		(*-----------------------Weiterschaltbedingungen----------------------------*)
		IF fb_bbgen_xml_file.fertig_lesen  AND NOT fb_state_entry.E THEN
			fb_state_entry.i16_next_step := 320;
		ELSIF fb_bbgen_xml_file.bError THEN
			sm_fehler_lesen_band := TRUE;
			fb_state_entry.i16_next_step := FEHLER;
		END_IF

(*=======================================================*)
	320:
		IF fb_state_entry.E THEN
			gst_datensatz_copy.st_band:= gst_datensatz.st_band ;
			fb_bbgen_xml_file.start_lesen_band := FALSE;
		END_IF

		(*-----------------------Weiterschaltbedingungen----------------------------*)
		IF hm_alle_daten_laden THEN
			fb_state_entry.i16_next_step := 350;
		ELSE
			IF gst_datensatz_copy.st_md.s_aktuelles_band<>gst_datensatz.st_md.s_aktuelles_band THEN
				fb_state_entry.i16_next_step := 880;
			ELSE
				fb_state_entry.i16_next_step := 999;
			END_IF
		END_IF

(*=======================================================*)
	350:	(* Wt Daten *)
		IF fb_state_entry.E THEN
			gst_datensatz.st_wt:=st_wt_leer;
		END_IF

		(*-----------------------Weiterschaltbedingungen----------------------------*)
		IF 	gst_datensatz.st_md.s_aktueller_wt <>'' THEN
			fb_state_entry.i16_next_step := 360;
		ELSIF 	hm_alle_daten_laden  THEN
				fb_state_entry.i16_next_step := 400;
			ELSE
				fb_state_entry.i16_next_step := 999;
		END_IF

	360:
		IF fb_state_entry.E THEN
			fb_bbgen_xml_file.start_lesen_wt := TRUE;
			fb_bbgen_xml_file.s_path := s_wt_path;
			fb_bbgen_xml_file.s_wt := gst_datensatz.st_md.s_aktueller_wt;
		END_IF

		(*-----------------------Weiterschaltbedingungen----------------------------*)
		IF fb_bbgen_xml_file.fertig_lesen  AND NOT fb_state_entry.E THEN
			fb_state_entry.i16_next_step := 370;
		ELSIF fb_bbgen_xml_file.bError THEN
			sm_fehler_lesen_wt := TRUE;
			fb_state_entry.i16_next_step := FEHLER;
		END_IF

(*=======================================================*)
	370:
		IF fb_state_entry.E THEN
			gst_datensatz_copy.st_wt:= gst_datensatz.st_wt ;
			fb_bbgen_xml_file.start_lesen_wt := FALSE;
		END_IF

		(*-----------------------Weiterschaltbedingungen----------------------------*)
		IF hm_alle_daten_laden THEN
			fb_state_entry.i16_next_step := 400;
		ELSE
			IF gst_datensatz_copy.st_md.s_aktueller_wt<>gst_datensatz.st_md.s_aktueller_wt THEN
				fb_state_entry.i16_next_step := 880;
			ELSE
				fb_state_entry.i16_next_step := 999;
			END_IF
		END_IF

(*=======================================================*)
	400:	(* Abfrage auf manuelle Anwahl des Bestückbildes *)
 		CASE gst_datensatz.st_md.i16_typ_bestueckmodus OF

			BESTUECKUNG_MANUAL:
				(* Bei der manuellen Auswahl des Bestückprogrammes werden die Daten direkt über die Visu
				von einem txt-File in die Variable "gst_datensatz" geladen. Ein Einlesen ist somit nicht nötig. *)
				gst_datensatz.st_bestueckprogramm:=gst_manuelles_bestueckprogramm;
				gst_datensatz.st_md.s_aktueller_isk:='ISK_Daten';
				IF hm_alle_daten_laden THEN
					fb_state_entry.i16_next_step := 600;
				ELSE
					fb_state_entry.i16_next_step := 999;
				END_IF

			BESTUECKUNG_HALBAUTO:
				IF gi16_maschinenstatusinfo = STATUS_MASCHINE_ARBEITET THEN
					gst_datensatz.st_md.s_aktueller_isk:='ISK_Daten';
					fb_state_entry.i16_next_step := 500;
				ELSE
					fb_state_entry.i16_next_step := 999;
				END_IF

			BESTUECKUNG_AUTO:
				IF gi16_maschinenstatusinfo = STATUS_MASCHINE_ARBEITET THEN
					fb_state_entry.i16_next_step := 410;
				ELSE
					fb_state_entry.i16_next_step := 999;
				END_IF

		END_CASE

(*=======================================================*)
	410:	(*alle Positonen löschen*)
		IF 	fb_state_entry.E THEN
			gst_bestueckbild := st_bestueckbild_leer;
			gst_datensatz.st_bestueckprogramm:=st_bestueckprogramm_leer;
		END_IF

		fb_state_entry.i16_next_step := 412;

(*=======================================================*)
	412:	(* Bestueckbild lesen und generieren *)
		IF fb_state_entry.E THEN
			fb_bbgen_xml_file.start_lesen_bestueckbild := TRUE;
			fb_bbgen_xml_file.s_path := s_bestueckbild_path;
			fb_bbgen_xml_file.s_bestueckbild := gst_datensatz.st_md.s_aktuelle_artikelnummer;
		END_IF

		(*-----------------------Weiterschaltbedingungen----------------------------*)
		IF fb_bbgen_xml_file.fertig_lesen  AND NOT fb_state_entry.E THEN
			IF	visu.b_merker_vollbestuecken THEN
				fb_state_entry.i16_next_step := 414;
			ELSE
				fb_state_entry.i16_next_step := 420;
			END_IF
		ELSIF fb_bbgen_xml_file.bError THEN
			sm_fehler_lesen_bestueckbild := TRUE;
			fb_state_entry.i16_next_step := FEHLER;
		END_IF

(*=======================================================*)
	414:	(* Werkzeuggruppen durchsuchen nach benuztem Werkzeug *)
		IF 	fb_state_entry.E THEN
			fb_bbgen_xml_file.start_lesen_bestueckbild := FALSE;
			i32_UsedTool:=-1;
			k:=-1;
			FOR k := 0 TO 4 DO
				i:=-1;

				FOR i := 0 TO MaxNoOfWkz DO
					IF 	gst_bestueckbild.s_wkzgruppe[k].s_wkznummer[i] = gst_datensatz.st_md.s_aktuelles_wkz THEN
						i32_UsedTool:=i;
					END_IF
				END_FOR
			END_FOR
		END_IF

		(*-----------------------Weiterschaltbedingungen----------------------------*)
		IF 	i32_UsedTool <> -1 THEN
			fb_state_entry.i16_next_step := 416;
		END_IF

		IF 	gst_bestueckbild.s_Bestueckbild_vollbestueckt[i32_UsedTool] = '' THEN
			fb_state_entry.i16_next_step := 420;
			bm_keine_vollbestueck_Artikelnummer:=TRUE;
		END_IF

(*=======================================================*)
	416:	(* Bestueckbild lesen und generieren *)
		IF fb_state_entry.E THEN
			fb_bbgen_xml_file.start_lesen_bestueckbild := TRUE;
			fb_bbgen_xml_file.s_path := s_bestueckbild_path;
			fb_bbgen_xml_file.s_bestueckbild := gst_bestueckbild.s_Bestueckbild_vollbestueckt[i32_UsedTool] ;
		END_IF

		(*-----------------------Weiterschaltbedingungen----------------------------*)
		IF fb_bbgen_xml_file.fertig_lesen  AND NOT fb_state_entry.E THEN
			fb_state_entry.i16_next_step := 420;
			fb_bbgen_xml_file.start_lesen_bestueckbild := FALSE;
		ELSIF fb_bbgen_xml_file.bError THEN
			sm_fehler_lesen_bestueckbild := TRUE;
			fb_state_entry.i16_next_step := FEHLER;
		END_IF

(*=======================================================*)
	420:	(* Generiere Bestückprogramm *)
		IF fb_state_entry.E THEN
			bm_kleinster_greifer_groesser_kleinste_pinanzahl_in_bb := FALSE;
			generiere_bestueckbild();
		END_IF

		(*-----------------------Weiterschaltbedingungen----------------------------*)
		fb_state_entry.i16_next_step := 425;

(*=======================================================*)
	425:	(* Hub_Faktor_ermitteln *)
		IF fb_state_entry.E THEN

			IF	gst_datensatz.st_wkz.i16_typ_bandeinzug=STANDARD_2FACH_V2  OR
				gst_datensatz.st_wkz.i16_typ_bandeinzug=BANDWECHSLER_V2 THEN
				Hub_Faktor_ermitteln();
			ELSE
				lr_FaktorHub:=1;
			END_IF

		END_IF

		(*-----------------------Weiterschaltbedingungen----------------------------*)
		fb_state_entry.i16_next_step := 430;

(*=======================================================*)
	430:	(* Schreibe Bestückprogramm auf HDD *)
		IF fb_state_entry.E THEN
			fb_bbgen_write_file.bStart := TRUE;
		END_IF


		(*-----------------------Weiterschaltbedingungen----------------------------*)
		IF NOT fb_state_entry.E THEN
			IF fb_bbgen_write_file.bFertig THEN
				fb_state_entry.i16_next_step := 600; (* ISK Daten lesen*)
			END_IF

			IF fb_bbgen_write_file.bError THEN
				fb_state_entry.i16_next_step := FEHLER;
				sm_fehler_schreiben_bestueckbild_auf_hdd := TRUE;
			END_IF
		END_IF

		IF fb_state_entry.X THEN
			fb_bbgen_write_file.bStart := FALSE;
		END_IF


(*=======================================================*)
	500:	(*alle Positonen löschen*)
		IF 	fb_state_entry.E THEN
			gst_bestueckbild_halbauto := st_bestueckbild_halbauto_leer;
		END_IF

		fb_state_entry.i16_next_step := 510;

(*=======================================================*)
	510:	(* halbauto Bestueckbild lesen  *)
		IF fb_state_entry.E THEN
			fb_bbgen_xml_file.start_lesen_bestueckbild_halbauto := TRUE;
			fb_bbgen_xml_file.s_path := s_bestueckbild_halbauto_path;
			fb_bbgen_xml_file.s_bestueckbild := gst_datensatz.st_md.s_aktuelle_artikelnummer;
		END_IF

		(*-----------------------Weiterschaltbedingungen----------------------------*)
		IF fb_bbgen_xml_file.fertig_lesen  AND NOT fb_state_entry.E THEN
			fb_state_entry.i16_next_step := 515;
		ELSIF fb_bbgen_xml_file.bError THEN
			sm_fehler_lesen_bestueckbild := TRUE;
			fb_state_entry.i16_next_step := FEHLER;
		END_IF

(*=======================================================*)
	515:	(* alle Positionen löschen  *)
		fb_bbgen_xml_file.start_lesen_bestueckbild_halbauto := FALSE;
		gst_datensatz.st_bestueckprogramm:=st_bestueckprogramm_leer;

		(*-----------------------Weiterschaltbedingungen----------------------------*)
		IF	b_Wkz_Gruppe_gebildet THEN
			fb_state_entry.i16_next_step := 540;
		ELSE
			fb_state_entry.i16_next_step := 520;
		END_IF

		IF	sm_Wkz_nicht_kompatibel OR
			sm_Wkz_Gruppe_nicht_zugeordnet THEN
			fb_state_entry.i16_next_step := FEHLER;
		END_IF

(*=======================================================*)
	520:	(* Werkzeuggruppen durchsuchen nach benuztem Werkzeug *)
		IF 	fb_state_entry.E THEN
			i32_UsedTool:=-1;
			k:=-1;
			FOR k := 0 TO 4 DO
				i:=-1;

				FOR i := 0 TO MaxNoOfWkz DO
					IF 	gst_bestueckbild_halbauto.s_wkzgruppe[k].s_wkznummer[i] = gst_datensatz.st_md.s_aktuelles_wkz THEN
						i32_UsedTool:=i;
					END_IF
				END_FOR
			END_FOR

		END_IF

		(*-----------------------Weiterschaltbedingungen----------------------------*)
		IF 	i32_UsedTool <> -1 THEN
			fb_state_entry.i16_next_step := 530;
		ELSE
			sm_fehler_wkz_nicht_vorhanden:=TRUE;
			fb_state_entry.i16_next_step := FEHLER;
		END_IF

(*=======================================================*)
	530: (*kopieren des zum WZ passenden Bestückbild*)
		IF 	fb_state_entry.E THEN
			gst_datensatz.st_bestueckprogramm:=gst_bestueckbild_halbauto.Wkz[i32_UsedTool];
			gst_datensatz.st_isk:=gst_bestueckbild_halbauto.Wkz[i32_UsedTool].st_isk;


			(*Offset dazurechnen*)
			k:=-1;
			FOR k := 0 TO (gst_bestueckbild_halbauto.Wkz[i32_UsedTool].i32_anzahl - 1) DO  (*max 511*)
				IF	gst_datensatz.st_bestueckprogramm.i16_b[k] = -1 THEN
					gst_datensatz.st_bestueckprogramm.lr_y[k]:=gst_datensatz.st_bestueckprogramm.lr_y[k] + gst_datensatz.st_bestueckprogramm.lr_y_offset;
					gst_datensatz.st_bestueckprogramm.lr_z[k]:=gst_datensatz.st_bestueckprogramm.lr_z[k] + gst_datensatz.st_bestueckprogramm.lr_z_offset;
				END_IF
			END_FOR

		END_IF

		(*-----------------------Weiterschaltbedingungen----------------------------*)
		IF 	gst_datensatz.st_bestueckprogramm.s_band = gst_datensatz.st_md.s_aktuelles_band  THEN
			fb_state_entry.i16_next_step := 590;
		ELSE
			sm_fehler_falsches_Band:=TRUE;
			fb_state_entry.i16_next_step := FEHLER;
		END_IF

(*=======================================================*)
(*Halbautomatisch mit Gruppen*)
	540:	(* prüfen ob Werkzeuggruppen gleiche Bänder haben *)
		IF 	fb_state_entry.E THEN

			k:=-1;
			FOR k := 0 TO 4 DO
				i:=-1;

				FOR i := 0 TO MaxNoOfWkz DO
					n:=-1;
					FOR n := 0 TO i16_anzahl_Wkz_Gruppen - 1 DO
						IF 	gst_bestueckbild_halbauto.s_wkzgruppe[k].s_wkznummer[i] = gst_datensatz.st_md.st_wkz_gruppe[n].s_wkz THEN
							gst_datensatz.st_md.st_wkz_gruppe[n].s_Band:=gst_bestueckbild_halbauto.Wkz[i].s_band;
							gst_datensatz.st_md.st_wkz_gruppe[n].i32_Anzahl:=gst_bestueckbild_halbauto.Wkz[i].i32_anzahl;
							gst_datensatz.st_md.st_wkz_gruppe[n].i32_Wkz_nr:=i;
						END_IF
					END_FOR

				END_FOR

			END_FOR

		END_IF


		i:=-1;
		b_Wkz_akt_vorhanden:=FALSE;
		FOR i := 0 TO i16_anzahl_Wkz_Gruppen - 1 DO
			IF	gst_datensatz.st_md.st_wkz_gruppe[i].s_Band <> '' AND
				gst_datensatz.st_md.st_wkz_gruppe[0].s_Band <> gst_datensatz.st_md.st_wkz_gruppe[i].s_Band THEN
				sm_Band_nicht_kompatibel:=TRUE;
			END_IF
			IF	gst_datensatz.st_md.s_aktuelles_wkz = gst_datensatz.st_md.st_wkz_gruppe[i].s_wkz THEN
				b_Wkz_akt_vorhanden:=TRUE;
			END_IF
		END_FOR
		sm_fehler_wkz_nicht_vorhanden:=NOT b_Wkz_akt_vorhanden;

		(*-----------------------Weiterschaltbedingungen----------------------------*)
		IF	sm_fehler_wkz_nicht_vorhanden OR
			sm_Band_nicht_kompatibel THEN
			fb_state_entry.i16_next_step := FEHLER;
		ELSE
			fb_state_entry.i16_next_step := 550;
		END_IF

(*=======================================================*)
	550: (*kopieren des zum WZ passenden Bestückbild*)
		IF 	fb_state_entry.E THEN
			i32_UsedTool:=gst_datensatz.st_md.st_wkz_gruppe[0].i32_Wkz_nr;
			gst_datensatz.st_bestueckprogramm:=gst_bestueckbild_halbauto.Wkz[i32_UsedTool];
			gst_datensatz.st_isk:=gst_bestueckbild_halbauto.Wkz[i32_UsedTool].st_isk;
			gst_datensatz.st_bestueckprogramm.i32_anzahl:=0;

			i:=-1;
			for_begin:=0;
			FOR i := 0 TO i16_anzahl_Wkz_Gruppen - 1 DO

				i32_UsedTool:=gst_datensatz.st_md.st_wkz_gruppe[i].i32_Wkz_nr;
				gst_datensatz.st_bestueckprogramm.i32_anzahl:=gst_datensatz.st_md.st_wkz_gruppe[i].i32_Anzahl + gst_datensatz.st_bestueckprogramm.i32_anzahl;

				for_end:=for_begin + gst_bestueckbild_halbauto.Wkz[i32_UsedTool].i32_anzahl - 1;

				FOR k := for_begin TO for_end DO  (*max 511*)
						gst_datensatz.st_bestueckprogramm.lr_y[k]:=		gst_bestueckbild_halbauto.Wkz[i32_UsedTool].lr_y[k - for_begin] + gst_bestueckbild_halbauto.Wkz[i32_UsedTool].lr_y_offset;
						gst_datensatz.st_bestueckprogramm.lr_z[k]:=		gst_bestueckbild_halbauto.Wkz[i32_UsedTool].lr_z[k - for_begin] + gst_bestueckbild_halbauto.Wkz[i32_UsedTool].lr_z_offset;
						gst_datensatz.st_bestueckprogramm.i16_b[k]:=	gst_bestueckbild_halbauto.Wkz[i32_UsedTool].i16_b[k - for_begin];
						gst_datensatz.st_bestueckprogramm.b_podest_verschieben[k]:=	gst_bestueckbild_halbauto.Wkz[i32_UsedTool].b_podest_verschieben[k - for_begin];
				END_FOR
				for_begin:=for_begin + gst_bestueckbild_halbauto.Wkz[i32_UsedTool].i32_anzahl ;

			END_FOR

		END_IF

		(*-----------------------Weiterschaltbedingungen----------------------------*)
		IF 	gst_datensatz.st_bestueckprogramm.s_band = gst_datensatz.st_md.s_aktuelles_band  THEN
			fb_state_entry.i16_next_step := 590;
		ELSE
			sm_fehler_falsches_Band:=TRUE;
			fb_state_entry.i16_next_step := FEHLER;
		END_IF

(*=======================================================*)
(*=======================================================*)
	590:	(* Hub_Faktor_ermitteln *)
		IF fb_state_entry.E THEN

			IF	gst_datensatz.st_wkz.i16_typ_bandeinzug=STANDARD_2FACH_V2 OR
				gst_datensatz.st_wkz.i16_typ_bandeinzug=BANDWECHSLER_V2 OR
				gst_datensatz.st_wkz.i16_typ_bandeinzug=SERVO THEN
				Hub_Faktor_ermitteln_halbauto();
			ELSE
				lr_FaktorHub:=1;
			END_IF

		END_IF

		(*-----------------------Weiterschaltbedingungen----------------------------*)
		fb_state_entry.i16_next_step := 999;

(*ISK Daten lesen===============================================*)
	600:
		IF fb_state_entry.E THEN
			fb_bbgen_xml_file.start_lesen_bestueckbild := FALSE;
			hm_alle_daten_laden:=FALSE;
		END_IF

		(*-----------------------Weiterschaltbedingungen----------------------------*)
		fb_state_entry.i16_next_step := 610;

(*=======================================================*)
	610:(* ISK Daten *)

		IF fb_state_entry.E THEN
			fb_bbgen_xml_file.start_lesen_isk := TRUE;
			fb_bbgen_xml_file.s_path := s_isk_path;
			fb_bbgen_xml_file.s_isk := gst_datensatz.st_md.s_aktueller_isk;
		END_IF

		(*-----------------------Weiterschaltbedingungen----------------------------*)
		IF fb_bbgen_xml_file.fertig_lesen  AND NOT fb_state_entry.E THEN
			fb_state_entry.i16_next_step := 620;
		ELSIF fb_bbgen_xml_file.bError THEN
			sm_fehler_lesen_isk := TRUE;
			fb_state_entry.i16_next_step := FEHLER;
		END_IF

(*=======================================================*)
	620:
		IF fb_state_entry.E THEN
			gst_datensatz_copy.st_isk:= gst_datensatz.st_isk ;
			fb_bbgen_xml_file.start_lesen_isk := FALSE;
		END_IF

		(*-----------------------Weiterschaltbedingungen----------------------------*)
		fb_state_entry.i16_next_step := 999;




(*===========================Speichern============================*)
	(* Alle aktuelle Daten von der Maschine und Werkzeug speichern *)
	800:	(* ISK daten *)
		IF fb_state_entry.E THEN
			fb_bbgen_xml_file.start_schreiben_isk := TRUE;
			fb_bbgen_xml_file.s_path := s_isk_path;
			fb_bbgen_xml_file.s_isk := gst_datensatz.st_md.s_aktueller_isk;
		END_IF

		(*-----------------------Weiterschaltbedingungen----------------------------*)
		IF fb_bbgen_xml_file.fertig_schreiben AND NOT fb_state_entry.E THEN
			fb_state_entry.i16_next_step := 810;
		ELSIF fb_bbgen_xml_file.bError THEN
			sm_fehler_schreiben_isk := TRUE;
			fb_state_entry.i16_next_step := FEHLER;
		END_IF

(*=======================================================*)
	810:
		IF fb_state_entry.E THEN
			gst_datensatz_copy.st_isk:= gst_datensatz.st_isk ;
			fb_bbgen_xml_file.start_schreiben_isk := FALSE;
		END_IF

		(*-----------------------Weiterschaltbedingungen----------------------------*)
		IF 	hm_alle_daten_speichern THEN
			fb_state_entry.i16_next_step := 820;
		ELSE
			fb_state_entry.i16_next_step := 999;
		END_IF

(*=======================================================*)
	820:	(* WKZ Daten *)
		IF (fb_state_entry.E) THEN
			fb_bbgen_xml_file.start_schreiben_wkz := TRUE;
			fb_bbgen_xml_file.s_path := s_wkz_path;
			fb_bbgen_xml_file.s_wkz := gst_datensatz.st_md.s_aktuelles_wkz;
		END_IF

		(*-----------------------Weiterschaltbedingungen----------------------------*)
		IF fb_bbgen_xml_file.fertig_schreiben  AND NOT fb_state_entry.E THEN
			fb_state_entry.i16_next_step := 830;
		ELSIF fb_bbgen_xml_file.bError THEN
			sm_fehler_schreiben_wkz := TRUE;
			fb_state_entry.i16_next_step := FEHLER;
		END_IF

(*=======================================================*)
	830:
		IF fb_state_entry.E THEN
			fb_bbgen_xml_file.start_schreiben_wkz := FALSE;
			gst_datensatz_copy.st_wkz:= gst_datensatz.st_wkz ;
		END_IF

		(*-----------------------Weiterschaltbedingungen----------------------------*)
		IF 	hm_alle_daten_speichern THEN
			fb_state_entry.i16_next_step := 840;
		ELSE
			fb_state_entry.i16_next_step := 999;
		END_IF

(*=======================================================*)
	840:	(* Band Daten *)
		IF (fb_state_entry.E) THEN
			fb_bbgen_xml_file.start_schreiben_band := TRUE;
			fb_bbgen_xml_file.s_path := s_band_path;
			fb_bbgen_xml_file.s_band := gst_datensatz.st_md.s_aktuelles_band;
		END_IF

		(*-----------------------Weiterschaltbedingungen----------------------------*)
		IF fb_bbgen_xml_file.fertig_schreiben  AND NOT fb_state_entry.E THEN
			fb_state_entry.i16_next_step := 850;
		ELSIF fb_bbgen_xml_file.bError THEN
			sm_fehler_schreiben_band := TRUE;
			fb_state_entry.i16_next_step := FEHLER;
		END_IF

(*=======================================================*)
	850:
		IF fb_state_entry.E THEN
			fb_bbgen_xml_file.start_schreiben_band := FALSE;
			gst_datensatz_copy.st_band:= gst_datensatz.st_band ;
		END_IF

		(*-----------------------Weiterschaltbedingungen----------------------------*)
		IF 	hm_alle_daten_speichern THEN
			fb_state_entry.i16_next_step := 860;
		ELSE
			fb_state_entry.i16_next_step := 999;
		END_IF

(*=======================================================*)
	860:	(* Wt Daten *)
		IF (fb_state_entry.E) THEN
			fb_bbgen_xml_file.start_schreiben_wt := TRUE;
			fb_bbgen_xml_file.s_path := s_wt_path;
			fb_bbgen_xml_file.s_wt := gst_datensatz.st_md.s_aktueller_wt;
		END_IF

		(*-----------------------Weiterschaltbedingungen----------------------------*)
		IF fb_bbgen_xml_file.fertig_schreiben  AND NOT fb_state_entry.E THEN
			fb_state_entry.i16_next_step := 870;
		ELSIF fb_bbgen_xml_file.bError THEN
			sm_fehler_schreiben_wt := TRUE;
			fb_state_entry.i16_next_step := FEHLER;
		END_IF

(*=======================================================*)
	870:
		IF fb_state_entry.E THEN
			fb_bbgen_xml_file.start_schreiben_wt := FALSE;
			gst_datensatz_copy.st_wt:= gst_datensatz.st_wt ;
		END_IF

		(*-----------------------Weiterschaltbedingungen----------------------------*)
		IF 	hm_alle_daten_speichern THEN
			fb_state_entry.i16_next_step := 880;
		ELSE
			fb_state_entry.i16_next_step := 999;
		END_IF

(*=======================================================*)
	880:	(* Maschinendaten *)
		IF (fb_state_entry.E) THEN
			fb_bbgen_xml_file.start_schreiben_md := TRUE;
			fb_bbgen_xml_file.s_path := s_md_path;
			fb_bbgen_xml_file.s_md := s_md_name;
		END_IF

		(*-----------------------Weiterschaltbedingungen----------------------------*)
		IF fb_bbgen_xml_file.fertig_schreiben  AND NOT fb_state_entry.E THEN
			fb_state_entry.i16_next_step := 882;
		ELSIF fb_bbgen_xml_file.bError THEN
			sm_fehler_schreiben_md := TRUE;
			fb_state_entry.i16_next_step := FEHLER;
		END_IF

	882:
		IF fb_state_entry.E THEN
			gst_datensatz_copy.st_md:= gst_datensatz.st_md ;
			fb_bbgen_xml_file.start_schreiben_md := FALSE;
			fb_state_entry.i16_next_step := 884;
		END_IF

	884:	(* Maschinendaten Backup *)
		IF (fb_state_entry.E) THEN
			fb_bbgen_xml_file.start_schreiben_md_backup := TRUE;
			fb_bbgen_xml_file.s_path := s_md_path;
			fb_bbgen_xml_file.s_md_backup := s_md_backup_name;
		END_IF

		(*-----------------------Weiterschaltbedingungen----------------------------*)
		IF fb_bbgen_xml_file.fertig_schreiben  AND NOT fb_state_entry.E THEN
			fb_state_entry.i16_next_step := 886;
		ELSIF fb_bbgen_xml_file.bError THEN
			sm_fehler_schreiben_md := TRUE;
			fb_state_entry.i16_next_step := FEHLER;
		END_IF

	886:
		IF fb_state_entry.E THEN
			fb_bbgen_xml_file.start_schreiben_md_backup := FALSE;
			fb_state_entry.i16_next_step := 999;
		END_IF

(*=======================================================*)
(* manuelle Bestückbilder in halbautomatische XML Dateien umwandeln
	->	PLC resetten (Strukturen leerern)
	->	Artikelnummer in MD eintragen ( Artikelnummer = XML Dateiname)
	->	Schritt 975 forcen
	->	manualle Bestückbilder nacheinader mit Visu vorne öffnen (mit der ersten beginnen)
		die Bestückbilder werden dann in die Struktur (Bestückbild halbauto) eingetragen
	->	Schritt 980 forcen = XML Datei wird erstellt ( D:\BBGen\BestueckbildHalbauto )
	->	in der XML Datei nicht vorhandene WZ löschen, Werkzeuge, Band, Beschreibung, Projekt eintragen
	->	neue XML Datei auf Server kopieren
*)
975:
	IF (fb_state_entry.E) THEN
		gst_manuelles_bestueckprogramm.i32_anzahl:=0;
		gst_manuelles_bestueckprogramm.s_band:='';
		gst_manuelles_bestueckprogramm.lr_y_offset:=0;
		gst_manuelles_bestueckprogramm.lr_z_offset:=0;

		k:=-1;
		FOR k := 0 TO 511 DO
			gst_manuelles_bestueckprogramm.lr_y[k]:=0;
			gst_manuelles_bestueckprogramm.lr_z[k]:=0;
			gst_manuelles_bestueckprogramm.i16_b[k]:=0;
		END_FOR
		gst_manuelles_bestueckprogramm_copy:=gst_manuelles_bestueckprogramm;
		wkz_Nr:=-1;
	END_IF

	fb_ton_wz(IN:= MEMCMP(ADR(gst_manuelles_bestueckprogramm_copy), ADR(gst_manuelles_bestueckprogramm), SIZEOF(gst_manuelles_bestueckprogramm_copy)) <> 0, PT:= t#600ms, Q=> , ET=> );

	IF	fb_ton_wz.Q  THEN
		wkz_Nr:=wkz_Nr+1;
		gst_bestueckbild_halbauto.Wkz[wkz_Nr]:=gst_manuelles_bestueckprogramm;
		gst_bestueckbild_halbauto.Wkz[wkz_Nr].st_isk:=gst_datensatz.st_isk;

		gst_manuelles_bestueckprogramm.i32_anzahl:=0;
		gst_manuelles_bestueckprogramm.s_band:='';
		gst_manuelles_bestueckprogramm.lr_y_offset:=0;
		gst_manuelles_bestueckprogramm.lr_z_offset:=0;

		k:=-1;
		FOR k := 0 TO 511 DO
			gst_manuelles_bestueckprogramm.lr_y[k]:=0;
			gst_manuelles_bestueckprogramm.lr_z[k]:=0;
			gst_manuelles_bestueckprogramm.i16_b[k]:=0;
		END_FOR

		gst_manuelles_bestueckprogramm_copy:=gst_manuelles_bestueckprogramm;
	END_IF

(*=======================================================*)
	980:	(* Bestückbild *)
		IF (fb_state_entry.E) THEN
			fb_bbgen_xml_file.start_schreiben_bestueckbild_halbauto := TRUE;
			fb_bbgen_xml_file.s_path := s_bestueckbild_halbauto_path;
			fb_bbgen_xml_file.s_bestueckbild := gst_datensatz.st_md.s_aktuelle_artikelnummer;
		END_IF

		(*-----------------------Weiterschaltbedingungen----------------------------*)
		IF fb_bbgen_xml_file.fertig_schreiben  AND NOT fb_state_entry.E THEN
			fb_state_entry.i16_next_step := 990;
		ELSIF fb_bbgen_xml_file.bError THEN
			sm_fehler_schreiben_bestueckbild := TRUE;
			fb_state_entry.i16_next_step := FEHLER;
		END_IF

(*=======================================================*)
	990:
		IF fb_state_entry.E THEN
			fb_bbgen_xml_file.start_schreiben_bestueckbild_halbauto := FALSE;
			fb_state_entry.i16_next_step := 999;
		END_IF

(*=======================================================*)
	999:	(* Ende - Befehl wurde korrekt abgearbeitet *)
		IF fb_state_entry.E THEN
			st_ctrl_out.b_fertig := TRUE;
			i16_auftrag := KEIN_BB_AUFTRAG;

			IF NOT b_lesen_komplett THEN
				gst_datensatz_copy := gst_datensatz;
			END_IF
			b_lesen_komplett:=TRUE;

			fb_state_entry.i16_next_step := 0;
		END_IF

(*=======================================================*)
	1000: (* Fehler *)
		IF fb_state_entry.E THEN
			st_ctrl_out.b_fehler := TRUE;
			fb_ton_quitt.IN := FALSE;
			fb_bbgen_xml_file.bQuit := FALSE;
		END_IF

		(*-----------------------Weiterschaltbedingungen----------------------------*)
		IF st_ctrl_in.b_quitt AND NOT fb_state_entry.E THEN
			st_ctrl_out.b_fehler := FALSE;
			fb_ton_quitt.IN := TRUE;
			fb_bbgen_xml_file.bQuit := TRUE;
		END_IF

		IF fb_ton_quitt.Q THEN
			fb_ton_quitt.IN := FALSE;
			fb_state_entry.i16_next_step := 0;
		END_IF
END_CASE

fb_state_entry(	i16_pos:= 2 );

(* ======================================Subkomponenten======================================== *)
fb_bbgen_xml_file(
	bQuit:= ,
	start_lesen_isk:= ,
	start_schreiben_isk:= ,
	start_lesen_wkz:= ,
	start_schreiben_wkz:= ,
	start_lesen_bestueckbild:= ,
	start_schreiben_bestueckbild:= ,
	start_lesen_md:= ,
	start_schreiben_md:= ,
	start_lesen_band:= ,
	start_schreiben_band:= ,
	s_path:= ,
	s_bestueckbild:= ,
	s_wkz:= ,
	s_isk:= ,
	s_md:= ,
	s_band:= ,
	fertig_lesen=> ,
	fertig_schreiben=> ,
	bError=> ,
	nErrId=> );

fb_bbgen_write_file(
	bStart:= ,
	bFertig=> ,
	bError=> );

fb_xml_srv_read(
	sNetId:= ,
	ePath:= PATH_GENERIC,
	nMode:= XMLSRV_SKIPMISSING,
	sSymName:= ,
	sFilePath:= ,
	sXPath:= ,
	bExecute:= ,
	tTimeout:= t#20s,
	bBusy=> ,
	bError=> ,
	nErrId=> );

IF st_config.b_config_fertig THEN
	garr_stoermeldungen[st_config.i16_meld_startindex + 0] := sm_fehler_lesen_band;
	garr_stoermeldungen[st_config.i16_meld_startindex + 1] := sm_fehler_lesen_bestueckbild;
	garr_stoermeldungen[st_config.i16_meld_startindex + 2] := sm_fehler_lesen_isk;
	garr_stoermeldungen[st_config.i16_meld_startindex + 3] := sm_fehler_lesen_md;
	garr_stoermeldungen[st_config.i16_meld_startindex + 4] := sm_fehler_lesen_wkz;
	garr_stoermeldungen[st_config.i16_meld_startindex + 5] := sm_fehler_schreiben_band;
	garr_stoermeldungen[st_config.i16_meld_startindex + 6] := sm_fehler_schreiben_bestueckbild;
	garr_stoermeldungen[st_config.i16_meld_startindex + 7] := sm_fehler_schreiben_isk;
	garr_stoermeldungen[st_config.i16_meld_startindex + 8] := sm_fehler_schreiben_md;
	garr_stoermeldungen[st_config.i16_meld_startindex + 9] := sm_fehler_schreiben_wkz;
	garr_stoermeldungen[st_config.i16_meld_startindex + 10] := sm_fehler_generieren_bestueckbild;
	garr_stoermeldungen[st_config.i16_meld_startindex + 11] := sm_fehler_schreiben_bestueckbild_auf_hdd;
	garr_stoermeldungen[st_config.i16_meld_startindex + 12] := sm_fehler_wkz_nicht_vorhanden;
	garr_stoermeldungen[st_config.i16_meld_startindex + 13] := sm_fehler_falsches_Band;
	garr_stoermeldungen[st_config.i16_meld_startindex + 14] := sm_Wkz_nicht_kompatibel;
	garr_stoermeldungen[st_config.i16_meld_startindex + 15] := sm_Band_nicht_kompatibel;
	garr_stoermeldungen[st_config.i16_meld_startindex + 16] := sm_Wkz_Gruppe_nicht_zugeordnet;
	garr_stoermeldungen[st_config.i16_meld_startindex + 17] := sm_fehler_lesen_wt;
	garr_stoermeldungen[st_config.i16_meld_startindex + 18] := sm_fehler_schreiben_wt;
	garr_stoermeldungen[st_config.i16_meld_startindex + 19] := FALSE;

	garr_betriebsmeldungen[st_config.i16_meld_startindex + 0] := bm_kleinster_greifer_groesser_kleinste_pinanzahl_in_bb;
	garr_betriebsmeldungen[st_config.i16_meld_startindex + 1] := bm_keine_vollbestueck_Artikelnummer;
	garr_betriebsmeldungen[st_config.i16_meld_startindex + 2] := FALSE;
	garr_betriebsmeldungen[st_config.i16_meld_startindex + 3] := FALSE;
	garr_betriebsmeldungen[st_config.i16_meld_startindex + 4] := FALSE;
	garr_betriebsmeldungen[st_config.i16_meld_startindex + 5] := FALSE;
	garr_betriebsmeldungen[st_config.i16_meld_startindex + 6] := FALSE;
	garr_betriebsmeldungen[st_config.i16_meld_startindex + 7] := FALSE;
	garr_betriebsmeldungen[st_config.i16_meld_startindex + 8] := FALSE;
	garr_betriebsmeldungen[st_config.i16_meld_startindex + 9] := FALSE;
	garr_betriebsmeldungen[st_config.i16_meld_startindex + 10] := FALSE;
	garr_betriebsmeldungen[st_config.i16_meld_startindex + 11] := FALSE;
	garr_betriebsmeldungen[st_config.i16_meld_startindex + 12] := FALSE;
	garr_betriebsmeldungen[st_config.i16_meld_startindex + 13] := FALSE;
	garr_betriebsmeldungen[st_config.i16_meld_startindex + 14] := FALSE;
	garr_betriebsmeldungen[st_config.i16_meld_startindex + 15] := FALSE;
	garr_betriebsmeldungen[st_config.i16_meld_startindex + 16] := FALSE;
	garr_betriebsmeldungen[st_config.i16_meld_startindex + 17] := FALSE;
	garr_betriebsmeldungen[st_config.i16_meld_startindex + 18] := FALSE;
	garr_betriebsmeldungen[st_config.i16_meld_startindex + 19] := FALSE;
END_IF
END_PROGRAM
ACTION auto_speichern_laden:
IF 	(MEMCMP(ADR(gst_datensatz_copy.st_md), ADR(gst_datensatz.st_md), SIZEOF(gst_datensatz_copy.st_md)) = 0 ) AND
	(MEMCMP(ADR(gst_datensatz_copy.st_wkz), ADR(gst_datensatz.st_wkz), SIZEOF(gst_datensatz_copy.st_wkz)) = 0 ) AND
	(MEMCMP(ADR(gst_datensatz_copy.st_band), ADR(gst_datensatz.st_band), SIZEOF(gst_datensatz_copy.st_band)) = 0 ) AND
	(MEMCMP(ADR(gst_datensatz_copy.st_wt), ADR(gst_datensatz.st_wt), SIZEOF(gst_datensatz_copy.st_wt)) = 0 ) AND
	(MEMCMP(ADR(gst_datensatz_copy.st_isk), ADR(gst_datensatz.st_isk), SIZEOF(gst_datensatz_copy.st_isk)) = 0 )
THEN
	hm_md_speichern:=FALSE;
END_IF

(*Bei einer Änderung der Wkz, des WT's oder Band Anwahl xml einlesen  *)
IF	b_lesen_komplett AND
	i16_auftrag = KEIN_BB_AUFTRAG AND
	NOT hm_md_speichern AND
	gst_datensatz_copy.st_md.s_aktuelles_wkz<>gst_datensatz.st_md.s_aktuelles_wkz THEN
	i16_auftrag:=LESE_WKZ;
	hm_md_speichern:=TRUE;
END_IF

IF	b_lesen_komplett AND
	i16_auftrag = KEIN_BB_AUFTRAG AND
	NOT hm_md_speichern AND
	gst_datensatz_copy.st_md.s_aktuelles_band<>gst_datensatz.st_md.s_aktuelles_band THEN
	i16_auftrag:=LESE_BAND;
	hm_md_speichern:=TRUE;
END_IF

IF	b_lesen_komplett AND
	i16_auftrag = KEIN_BB_AUFTRAG AND
	NOT hm_md_speichern AND
	gst_datensatz_copy.st_md.s_aktueller_wt<>gst_datensatz.st_md.s_aktueller_wt THEN
	i16_auftrag:=LESE_WT;
	hm_md_speichern:=TRUE;
END_IF

(* Beim Umschalten auf Manuell ISK einlesen und Bestückbild zuweisen  *)
IF	b_lesen_komplett AND
	i16_auftrag = KEIN_BB_AUFTRAG AND
	NOT hm_md_speichern THEN
	fb_r_trig_taste_bestueckprg_manuell(CLK:= gst_datensatz.st_md.i16_typ_bestueckmodus=BESTUECKUNG_MANUAL, Q=> );

	IF	fb_r_trig_taste_bestueckprg_manuell.Q THEN
		gst_datensatz.st_md.s_aktueller_isk:='ISK_Daten';
		gst_datensatz.st_bestueckprogramm:=gst_manuelles_bestueckprogramm;
		i16_auftrag:=SCHREIBE_ISK;
		hm_md_speichern:=TRUE;
	END_IF
END_IF

(*=======================================================================================*)
(*Bei einer Änderung automatisch speichern===================================================*)

(*Ausnahmen*)
IF	b_lesen_komplett AND
	(MEMCMP(ADR(gst_datensatz_copy.st_isk), ADR(gst_datensatz.st_isk), SIZEOF(gst_datensatz_copy.st_isk)) <> 0 )  OR
	gst_datensatz_copy.st_md.i32_bestueckhubzaehler<>gst_datensatz.st_md.i32_bestueckhubzaehler OR
	(MEMCMP(ADR(gst_datensatz_copy.st_stueckzahlen), ADR(gst_datensatz.st_stueckzahlen), SIZEOF(gst_datensatz_copy.st_stueckzahlen)) <> 0 ) THEN
	gst_datensatz_copy.st_stueckzahlen:=gst_datensatz.st_stueckzahlen;
(*	gst_datensatz_copy.st_isk:=gst_datensatz.st_isk*);
END_IF

(*========================================================================================*)
(*ohne Timer wurde nicht immer gespeichert*)
fb_ton_end(
	IN:=  i16_auftrag = KEIN_BB_AUFTRAG AND b_lesen_komplett,
	PT:= t#100ms,
	Q=> ,
	ET=> );


(*Isk Daten speichern*)
IF	fb_ton_end.Q AND
	gst_datensatz.st_md.i16_typ_bestueckmodus=BESTUECKUNG_MANUAL AND
	(MEMCMP(ADR(gst_datensatz_copy.st_isk), ADR(gst_datensatz.st_isk), SIZEOF(gst_datensatz_copy.st_isk)) <> 0 ) THEN
	gst_datensatz_copy.st_isk:= gst_datensatz.st_isk ;
	i16_auftrag:=SCHREIBE_ISK;	(*ISK soll nur vom UML Designer verändert werden*)
END_IF

(*Nocken speichern und Rest ignorieren*)
IF	fb_ton_end.Q AND
	(MEMCMP(ADR(gst_datensatz_copy.st_wkz.nockenschaltwerk_bestueckachse), ADR(gst_datensatz.st_wkz.nockenschaltwerk_bestueckachse), SIZEOF(gst_datensatz_copy.st_wkz.nockenschaltwerk_bestueckachse)) <> 0 ) THEN
	FOR j := 0 TO MAX_NOCKENGERUEST DO	(*nur die Nocken begin und end speichern*)
		IF	gst_datensatz_copy.st_wkz.nockenschaltwerk_bestueckachse.arr_nocken[j].r_cam_begin<>gst_datensatz.st_wkz.nockenschaltwerk_bestueckachse.arr_nocken[j].r_cam_begin OR
			gst_datensatz_copy.st_wkz.nockenschaltwerk_bestueckachse.arr_nocken[j].r_cam_end<>gst_datensatz.st_wkz.nockenschaltwerk_bestueckachse.arr_nocken[j].r_cam_end THEN
			i16_auftrag:=SCHREIBE_WKZ;
		END_IF
	END_FOR
	gst_datensatz_copy.st_wkz.nockenschaltwerk_bestueckachse:=gst_datensatz.st_wkz.nockenschaltwerk_bestueckachse;
END_IF

(*Wkz Daten speichern*)
IF	fb_ton_end.Q AND
	gi16_maschinenstatusinfo <> STATUS_MASCHINE_ARBEITET AND
	(MEMCMP(ADR(gst_datensatz_copy.st_wkz), ADR(gst_datensatz.st_wkz), SIZEOF(gst_datensatz_copy.st_wkz)) <> 0 ) THEN
	i16_auftrag:=SCHREIBE_WKZ;
END_IF

(*Band Daten speichern*)
IF	fb_ton_end.Q AND
	gi16_maschinenstatusinfo <> STATUS_MASCHINE_ARBEITET AND
	(MEMCMP(ADR(gst_datensatz_copy.st_band), ADR(gst_datensatz.st_band), SIZEOF(gst_datensatz_copy.st_band)) <> 0 ) THEN
	i16_auftrag:=SCHREIBE_BAND;
END_IF

(*Wt Daten speichern*)
IF	fb_ton_end.Q AND
	gi16_maschinenstatusinfo <> STATUS_MASCHINE_ARBEITET AND
	(MEMCMP(ADR(gst_datensatz_copy.st_wt), ADR(gst_datensatz.st_wt), SIZEOF(gst_datensatz_copy.st_wt)) <> 0 ) THEN
	i16_auftrag:=SCHREIBE_WT;
END_IF

(*Maschinen Daten speichern*)
IF	fb_ton_end.Q AND
	gi16_maschinenstatusinfo <> STATUS_MASCHINE_ARBEITET AND
	(MEMCMP(ADR(gst_datensatz_copy.st_md), ADR(gst_datensatz.st_md), SIZEOF(gst_datensatz_copy.st_md)) <> 0 ) THEN
	i16_auftrag:=SCHREIBE_MD;
	hm_md_speichern:=FALSE;
END_IF
END_ACTION
ACTION generiere_bestueckbild:
(* Step 1: erzeuge eine Liste mit allen unseren Pins *)
st_akt_bestueckprogramm.i32_anzahl := 0;

FOR i := 0 TO gst_bestueckbild.i32_anzahl_pins - 1 BY 1
DO
	IF (gst_bestueckbild.st_pins[i].typ = gst_datensatz.st_md.s_aktuelles_band) THEN
		st_akt_bestueckprogramm.lr_y[st_akt_bestueckprogramm.i32_anzahl] := gst_bestueckbild.st_pins[i].lr_y;
		st_akt_bestueckprogramm.lr_z[st_akt_bestueckprogramm.i32_anzahl] := gst_bestueckbild.st_pins[i].lr_z;
		st_akt_bestueckprogramm.i16_b[st_akt_bestueckprogramm.i32_anzahl] := 1;

		st_akt_bestueckprogramm.i32_anzahl  := st_akt_bestueckprogramm.i32_anzahl + 1;
	END_IF
END_FOR


(* Step 2: Sortieren: Bubblesort by Z *)
sort_akt();

(* Einragen in die globale Sruktur *)
gst_datensatz.st_bestueckprogramm := st_akt_bestueckprogramm;
gst_datensatz.st_md.s_aktueller_isk := gst_bestueckbild.s_isknummer;
END_ACTION
ACTION Hub_Faktor_ermitteln:
 (*ermitteln der maximal zu bestückenden Pins eines Bestückbildes=========================*)

FOR n := 0 TO 14 DO
	s_HelpBand[n]:='';
	i32_Anzahl[n]:=0;
END_FOR
i32_maxAnzahl := 0;

FOR n := 0 TO 14 DO
	FOR m := 0 TO gst_bestueckbild.i32_anzahl_pins - 1 DO
		IF	gst_bestueckbild.st_pins[m].typ <> s_HelpBand[0] AND
			gst_bestueckbild.st_pins[m].typ <> s_HelpBand[1] AND
			gst_bestueckbild.st_pins[m].typ <> s_HelpBand[2] AND
			gst_bestueckbild.st_pins[m].typ <> s_HelpBand[3] AND
			gst_bestueckbild.st_pins[m].typ <> s_HelpBand[4] AND
			gst_bestueckbild.st_pins[m].typ <> s_HelpBand[5] AND
			gst_bestueckbild.st_pins[m].typ <> s_HelpBand[6] AND
			gst_bestueckbild.st_pins[m].typ <> s_HelpBand[7] AND
			gst_bestueckbild.st_pins[m].typ <> s_HelpBand[8] AND
			gst_bestueckbild.st_pins[m].typ <> s_HelpBand[9] AND
			gst_bestueckbild.st_pins[m].typ <> s_HelpBand[10] AND
			gst_bestueckbild.st_pins[m].typ <> s_HelpBand[11] AND
			gst_bestueckbild.st_pins[m].typ <> s_HelpBand[12] AND
			gst_bestueckbild.st_pins[m].typ <> s_HelpBand[13] AND
			gst_bestueckbild.st_pins[m].typ <> s_HelpBand[14] THEN
			s_HelpBand[n]:=gst_bestueckbild.st_pins[m].typ;
		END_IF
	END_FOR
END_FOR

FOR n := 0 TO 14 DO
	FOR m := 0 TO gst_bestueckbild.i32_anzahl_pins - 1 DO
		IF gst_bestueckbild.st_pins[m].typ = s_HelpBand[n] AND s_HelpBand[n] <>'' THEN
			i32_Anzahl[n]:=i32_Anzahl[n]+1;
		END_IF
	END_FOR
	IF	i32_Anzahl[n]>i32_maxAnzahl THEN
		i32_maxAnzahl:=i32_Anzahl[n];
	END_IF
END_FOR

(* Faktor für die Hubzahl*)
lr_min_FaktorHub:=100/gst_datensatz.st_wkz.r_auto;

IF	i32_maxAnzahl > 0  THEN

	lr_FaktorHub:=(DINT_TO_LREAL(st_akt_bestueckprogramm.i32_anzahl) / DINT_TO_LREAL(i32_maxAnzahl)) * 1.2;
	IF	lr_FaktorHub > 1 THEN
		lr_FaktorHub:=1;
	END_IF
	IF	lr_FaktorHub < lr_min_FaktorHub THEN 	(*Bestückgeschwindigkeit nur um maximal 100Hub verringern*)
		lr_FaktorHub:=lr_min_FaktorHub;
	END_IF
ELSE
	lr_FaktorHub:=1;
END_IF
END_ACTION
ACTION Hub_Faktor_ermitteln_halbauto:
 (*ermitteln der maximal zu bestückenden Pins eines Bestückbildes=========================*)
n:=-1;
i32_maxAnzahl := 0;
FOR n := 0 TO 14 DO
	i32_Anzahl[n]:=gst_bestueckbild_halbauto.Wkz[n].i32_anzahl;
	IF	i32_Anzahl[n]>i32_maxAnzahl THEN
		i32_maxAnzahl:=i32_Anzahl[n];
	END_IF
END_FOR

(* Faktor für die Hubzahl*)
lr_min_FaktorHub:=100/gst_datensatz.st_wkz.r_auto;

IF	i32_maxAnzahl > 0  THEN

	lr_FaktorHub:=(DINT_TO_LREAL(gst_datensatz.st_bestueckprogramm.i32_anzahl) / DINT_TO_LREAL(i32_maxAnzahl)) * 1.35;
	IF	lr_FaktorHub > 1 THEN
		lr_FaktorHub:=1;
	END_IF
	IF	lr_FaktorHub < lr_min_FaktorHub THEN 	(*Bestückgeschwindigkeit nur um maximal 100Hub verringern*)
		lr_FaktorHub:=lr_min_FaktorHub;
	END_IF
ELSE
	lr_FaktorHub:=1;
END_IF
END_ACTION
ACTION path:
IF	s_Projekt_path <> '' THEN
	IF	FIND(s_md_path,':') = 0 THEN
		s_md_path 	:= CONCAT(s_Projekt_path,s_md_path);
	END_IF
	IF	FIND(s_tools_path,':') = 0 THEN
		s_tools_path 	:= CONCAT(s_Projekt_path,s_tools_path);
	END_IF
END_IF
END_ACTION
ACTION sort_akt:
FOR i := st_akt_bestueckprogramm.i32_anzahl -1 TO 1  BY -1
DO
	FOR k := 0 TO i -1 BY 1
	DO
		CASE gst_bestueckbild.enu_richtung OF

			(* Y Spalte Minus nach Plus: Bei gleichem Y: Z minus nach Plus *)
			YMinus_nach_YPlus_ZMinus_nach_ZPlus:
				IF F_Vergleich_LReal(st_akt_bestueckprogramm.lr_y[k+1] , st_akt_bestueckprogramm.lr_y[k]) THEN
					b_sort_swap := st_akt_bestueckprogramm.lr_z[k+1] < st_akt_bestueckprogramm.lr_z[k];
				ELSE
					b_sort_swap := st_akt_bestueckprogramm.lr_y[k+1] < st_akt_bestueckprogramm.lr_y[k];
				END_IF

			(* Y Spalte Minus nach Plus: Bei gleichem Y: Z Plus nach Minus *)
			YMinus_nach_YPlus_ZPlus_nach_ZMinus:
				IF F_Vergleich_LReal(st_akt_bestueckprogramm.lr_y[k+1] , st_akt_bestueckprogramm.lr_y[k]) THEN
					b_sort_swap := st_akt_bestueckprogramm.lr_z[k+1] > st_akt_bestueckprogramm.lr_z[k];
				ELSE
					b_sort_swap := st_akt_bestueckprogramm.lr_y[k+1]< st_akt_bestueckprogramm.lr_y[k];
				END_IF

			(* Y Spalte Plus nach Minus: Bei gleichem Y: Z Minus nach Plus *)
			YPlus_nach_YMinus_ZMinus_nach_ZPlus:
				IF F_Vergleich_LReal(st_akt_bestueckprogramm.lr_y[k+1] , st_akt_bestueckprogramm.lr_y[k]) THEN
					b_sort_swap := st_akt_bestueckprogramm.lr_z[k+1] < st_akt_bestueckprogramm.lr_z[k];
				ELSE
					b_sort_swap := st_akt_bestueckprogramm.lr_y[k+1] > st_akt_bestueckprogramm.lr_y[k];
				END_IF

			(* Y Spalte Plus nach Minus: Bei gleichem Y: Z Plus nach Minus *)
			YPlus_nach_YMinus_ZPlus_nach_ZMinus:
				IF F_Vergleich_LReal(st_akt_bestueckprogramm.lr_y[k+1] , st_akt_bestueckprogramm.lr_y[k]) THEN
					b_sort_swap := st_akt_bestueckprogramm.lr_z[k+1] > st_akt_bestueckprogramm.lr_z[k];
				ELSE
					b_sort_swap := st_akt_bestueckprogramm.lr_y[k+1] > st_akt_bestueckprogramm.lr_y[k];
				END_IF
		END_CASE

		IF b_sort_swap THEN
			(* Tauschen k + 1 <--> k *)
			swap_a := k; swap_b := k+1;	swap_in_akt();
		END_IF

	END_FOR
END_FOR
END_ACTION
ACTION subr_Wkz_Band_Wt_schreiben:
(* ======================================Schrittkette======================================== *)
fb_state_entry2(	i16_pos:= 1 );

CASE fb_state_entry2.i16_step OF
(*=======================================================*)
	0:

		fb_wkz_band_wt_schreiben.Start := FALSE;

		(*-----------------------Weiterschaltbedingungen----------------------------*)
		fb_state_entry2.i16_next_step := BEREIT;

(*=======================================================*)
	BEREIT:	(* Warte auf Änderung *)

		(*-----------------------Weiterschaltbedingungen----------------------------*)
		IF gst_datensatz.st_md.s_aktuelles_wkz <> s_name_alt_wkz OR
		    gst_datensatz.st_md.s_aktuelles_band <> s_name_alt_band OR
		    gst_datensatz.st_md.s_aktueller_wt <> s_name_alt_wt THEN
			s_name_alt_wkz := gst_datensatz.st_md.s_aktuelles_wkz;
			s_name_alt_band :=gst_datensatz.st_md.s_aktuelles_band;
			s_name_alt_wt := gst_datensatz.st_md.s_aktueller_wt;
			fb_state_entry2.i16_next_step := 200;
		END_IF

(*=======================================================*)
	200: (* Aktuelles WKZ in txt Datei schreiben *)
		IF fb_state_entry2.E THEN
			fb_wkz_band_wt_schreiben.ExportStr := gst_datensatz.st_md.s_aktuelles_wkz;
			fb_wkz_band_wt_schreiben.FileName := 'Aktuelles_Wkz.txt';
			fb_wkz_band_wt_schreiben.Start := TRUE;
		END_IF

		(*-----------------------Weiterschaltbedingungen----------------------------*)
		IF fb_wkz_band_wt_schreiben.Busy THEN
			fb_wkz_band_wt_schreiben.Start := FALSE;
			fb_state_entry2.i16_next_step := 210;
		END_IF

(*=======================================================*)
	210: (* warte auf fertig *)

		(*-----------------------Weiterschaltbedingungen----------------------------*)
		IF fb_wkz_band_wt_schreiben.Done THEN
			fb_state_entry2.i16_next_step := 300;
		END_IF

(*=======================================================*)
	300: (* Aktuelles WKZ in txt Datei schreiben *)
		IF fb_state_entry2.E THEN
			fb_wkz_band_wt_schreiben.ExportStr := gst_datensatz.st_md.s_aktuelles_band;
			fb_wkz_band_wt_schreiben.FileName := 'Aktuelles_Band.txt';
			fb_wkz_band_wt_schreiben.Start := TRUE;
		END_IF

		(*-----------------------Weiterschaltbedingungen----------------------------*)
		IF fb_wkz_band_wt_schreiben.Busy THEN
			fb_wkz_band_wt_schreiben.Start := FALSE;
			fb_state_entry2.i16_next_step := 310;
		END_IF

(*=======================================================*)
	310: (* warte auf fertig *)

		(*-----------------------Weiterschaltbedingungen----------------------------*)
		IF fb_wkz_band_wt_schreiben.Done THEN
			fb_state_entry2.i16_next_step := 400;
		END_IF

(*=======================================================*)
	400: (* Aktuellen Wt in txt Datei schreiben *)
		IF fb_state_entry2.E THEN
			fb_wkz_band_wt_schreiben.ExportStr := gst_datensatz.st_md.s_aktueller_wt;
			fb_wkz_band_wt_schreiben.FileName := 'Aktueller_Wt.txt';
			fb_wkz_band_wt_schreiben.Start := TRUE;
		END_IF

		(*-----------------------Weiterschaltbedingungen----------------------------*)
		IF fb_wkz_band_wt_schreiben.Busy THEN
			fb_wkz_band_wt_schreiben.Start := FALSE;
			fb_state_entry2.i16_next_step := 410;
		END_IF

(*=======================================================*)
	410: (* warte auf fertig *)

		(*-----------------------Weiterschaltbedingungen----------------------------*)
		IF fb_wkz_band_wt_schreiben.Done THEN
			fb_state_entry2.i16_next_step := BEREIT;
		END_IF

END_CASE

fb_state_entry2(i16_pos:= 2 );

fb_wkz_band_wt_schreiben(
	Start:= ,
	ExportStr:= ,
	FileName:= ,
	Path:= 'D:\BBgen\',
	Mode:= 2,
	Ready=> , 
	Busy=> , 
	Done=> ,
	Error=> );
END_ACTION
ACTION swap_in_akt:
lr_tmp := st_akt_bestueckprogramm.lr_y[swap_a];
st_akt_bestueckprogramm.lr_y[swap_a] := st_akt_bestueckprogramm.lr_y[swap_b];
st_akt_bestueckprogramm.lr_y[swap_b] := lr_tmp;

lr_tmp := st_akt_bestueckprogramm.lr_z[swap_a];
st_akt_bestueckprogramm.lr_z[swap_a] := st_akt_bestueckprogramm.lr_z[swap_b];
st_akt_bestueckprogramm.lr_z[swap_b] := lr_tmp;

i16_tmp := st_akt_bestueckprogramm.i16_b[swap_a];
st_akt_bestueckprogramm.i16_b[swap_a] := st_akt_bestueckprogramm.i16_b[swap_b];
st_akt_bestueckprogramm.i16_b[swap_b] := i16_tmp;
END_ACTION
ACTION wkz_gruppe_kompatibel:
(*Gruppe löschen wenn ein neues Werkzeug ausgewählt wird*)
IF	gst_datensatz_copy.st_md.s_aktuelles_wkz<>gst_datensatz.st_md.s_aktuelles_wkz THEN
	i:=-1;
	FOR i := 0 TO 4 DO
		gst_datensatz.st_md.st_wkz_gruppe[i].s_wkz := '';
		gst_datensatz.st_md.st_wkz_gruppe[i].i16_wkz_gruppe_kompatibel := 0;
		gst_datensatz.st_md.st_wkz_gruppe[i].s_Band := '';
		gst_datensatz.st_md.st_wkz_gruppe[i].i32_Wkz_nr := -1;
		gst_datensatz.st_md.st_wkz_gruppe[i].i32_Anzahl := -1;
	END_FOR
END_IF

(*Fehler*)
IF	state =0 THEN
	k:=-1;
	sm_Wkz_Gruppe_nicht_zugeordnet:=FALSE;
	sm_Wkz_nicht_kompatibel:=FALSE;
	FOR k := 0 TO 4 DO
		i:=-1;
		FOR i := 0 TO 4 DO
			IF	gst_datensatz.st_md.st_wkz_gruppe[k].s_wkz <> '' AND
				gst_datensatz.st_md.st_wkz_gruppe[i].s_wkz <> '' AND
				gst_datensatz.st_md.st_wkz_gruppe[k].i16_wkz_gruppe_kompatibel <>gst_datensatz.st_md.st_wkz_gruppe[i].i16_wkz_gruppe_kompatibel THEN
				sm_Wkz_nicht_kompatibel:=TRUE;
			END_IF
		END_FOR

		IF	gst_datensatz.st_md.st_wkz_gruppe[k].s_wkz <> '' AND
			gst_datensatz.st_md.st_wkz_gruppe[k].i16_wkz_gruppe_kompatibel = 0 THEN
			sm_Wkz_Gruppe_nicht_zugeordnet:=TRUE;
		END_IF

	END_FOR
END_IF

(*==========================================================================================*)
b_Wkz_Gruppe_gebildet:=
	NOT sm_Wkz_nicht_kompatibel AND
	gst_datensatz.st_md.st_wkz_gruppe[0].s_wkz <> '' AND
	gst_datensatz.st_md.st_wkz_gruppe[1].s_wkz <> '';

i16_anzahl_Wkz_Gruppen:=0;
k:=-1;
FOR k := 0 TO 4 DO
	IF	gst_datensatz.st_md.st_wkz_gruppe[k].s_wkz <> ''	THEN
		i16_anzahl_Wkz_Gruppen:=i16_anzahl_Wkz_Gruppen + 1;
	END_IF
END_FOR

(*==========================================================================================*)
CASE state OF
0:	(* Auslesen wenn ein neues Wkz ausgewählt wird*)
	fb_xml_srv_read.bExecute:= FALSE;
	k:=-1;
	FOR k := 0 TO 4 DO
		IF	state =0 AND
			st_wkz_gruppe_copy[k].s_wkz<>gst_datensatz.st_md.st_wkz_gruppe[k].s_wkz THEN

			IF	gst_datensatz.st_md.st_wkz_gruppe[k].s_wkz='' THEN
				st_wkz_gruppe_copy[k].s_wkz:=gst_datensatz.st_md.st_wkz_gruppe[k].s_wkz;
			ELSE
				i32_neues_Wkz:=k;
				state:=10;
			END_IF

			gst_datensatz.st_md.st_wkz_gruppe[k].i16_wkz_gruppe_kompatibel:=0;
			st_wkz_gruppe_copy[k].i16_wkz_gruppe_kompatibel:=0;
			gst_datensatz.st_md.st_wkz_gruppe[k].s_Band := '';
			gst_datensatz.st_md.st_wkz_gruppe[k].i32_Wkz_nr := -1;
			gst_datensatz.st_md.st_wkz_gruppe[k].i32_Anzahl := -1;

		END_IF
	END_FOR

10:	(*Start auslesen*)
	nErrId := 0;
	fb_xml_srv_read.sFilePath:= 'D:\BBgen\Wkz\';
	fb_xml_srv_read.sFilePath:= CONCAT(fb_xml_srv_read.sFilePath,gst_datensatz.st_md.st_wkz_gruppe[i32_neues_Wkz].s_wkz);
	fb_xml_srv_read.sFilePath:= CONCAT(fb_xml_srv_read.sFilePath,'.xml');
	fb_xml_srv_read.sXPath := '/root/gst_datensatz.st_wkz/I16_WKZ_GRUPPE_KOMPATIBEL';
	fb_xml_srv_read.sSymName:= '.gst_datensatz.st_md.st_wkz_gruppe[';
	fb_xml_srv_read.sSymName:= CONCAT(fb_xml_srv_read.sSymName,DINT_TO_STRING(i32_neues_Wkz));
	fb_xml_srv_read.sSymName:= CONCAT(fb_xml_srv_read.sSymName,'].i16_wkz_gruppe_kompatibel');
	fb_xml_srv_read.bExecute:= TRUE;

	IF fb_xml_srv_read.bBusy THEN
		fb_xml_srv_read.bExecute:= FALSE;
		state := 20;
	END_IF

20:	(* Lesevorgang erfolgreich? *)
	IF NOT fb_xml_srv_read.bBusy THEN
		IF NOT fb_xml_srv_read.bError THEN
			state := 0;
			st_wkz_gruppe_copy[i32_neues_Wkz].s_wkz:=gst_datensatz.st_md.st_wkz_gruppe[i32_neues_Wkz].s_wkz;
			st_wkz_gruppe_copy[i32_neues_Wkz].i16_wkz_gruppe_kompatibel:=gst_datensatz.st_md.st_wkz_gruppe[i32_neues_Wkz].i16_wkz_gruppe_kompatibel;
		ELSE	(* Fehler *)
			nErrId := fb_xml_srv_read.nErrId;
			state := FEHLER;
		END_IF
	END_IF

FEHLER:
	state := 0;
	st_wkz_gruppe_copy[i32_neues_Wkz].s_wkz:=gst_datensatz.st_md.st_wkz_gruppe[i32_neues_Wkz].s_wkz;
END_CASE
END_ACTION

(* POU Gemeinsamkeiten17xx/BBGen/ST_BBGenXMLFile, ST *)
FUNCTION_BLOCK ST_BBGenXMLFile
VAR_INPUT
	bQuit								: BOOL;
	(* ISK *)
	start_lesen_isk						: BOOL;
	start_schreiben_isk					: BOOL;

	(* Wkz *)
	start_lesen_wkz						: BOOL;
	start_schreiben_wkz					: BOOL;

	(* Bestueckbild wird nur gelesen *)
	start_lesen_bestueckbild				: BOOL;
	start_schreiben_bestueckbild			: BOOL;

	(* Bestueckbild Halbautomatik wird nur gelesen *)
	start_lesen_bestueckbild_halbauto				: BOOL;
	start_schreiben_bestueckbild_halbauto			: BOOL;

	(* Maschinendaten *)
	start_lesen_md						: BOOL;
	start_schreiben_md					: BOOL;
	start_schreiben_md_backup			: BOOL;

	(* Banddaten *)
	start_lesen_band						: BOOL;
	start_schreiben_band					: BOOL;

	(* Wt-Daten *)
	start_lesen_wt						: BOOL;
	start_schreiben_wt						: BOOL;

	(* Wo liegen die Dateien *)
	s_path								: STRING(255);

	(* Welche Dateien? *)
	s_bestueckbild						: STRING(50);
	s_wkz								: STRING(50);
	s_isk								: STRING(50);
	s_md								: STRING(50);
	s_md_backup						: STRING(50);
	s_band								: STRING(50);
	s_wt									: STRING(50);
END_VAR
VAR_OUTPUT
	fertig_lesen							: BOOL;
	fertig_schreiben						: BOOL;

	bError								: BOOL;
	nErrId								: UDINT;
END_VAR
VAR
	fb_state_entry							: ST_StateEntry;
	fb_ton_quitt							: TON;
	fb_xml_srv_write						: FB_XmlSrvWriteByName;
	fb_xml_srv_read						: FB_XmlSrvReadByName;
	s_file								: STRING(255);

END_VAR
fb_ton_quitt(IN:= , PT:= t#50ms, Q=> , ET=> );

(* ======================================Schrittkette======================================== *)
fb_state_entry(
	i16_next_step:= ,
	i16_pos:= 1,
	s_debugtext:= ,
	E=> ,
	X=> ,
	i16_step=> ,
	i16_last_step=> );


CASE fb_state_entry.i16_step OF
(*=======================================================*)
	0:
		bError := FALSE;
		nErrId := 0;

		fertig_lesen := FALSE;
		fertig_schreiben := FALSE;

		fb_state_entry.i16_next_step := 10;

(*=======================================================*)
	10:	(* Auslesen der Daten aus den XML-Files *)
		(* Daten lesen *)
		IF start_lesen_isk THEN
			s_file := CONCAT(s_path, s_isk);
			s_file := CONCAT(s_file,'.xml');
			fb_xml_srv_read.sSymName := '.gst_datensatz.st_isk';
			fb_xml_srv_read.sXPath := '/root/gst_datensatz.st_isk';
			fb_state_entry.i16_next_step := 100;
		ELSIF start_lesen_bestueckbild THEN
			s_file := CONCAT(s_path, s_bestueckbild);
			s_file := CONCAT(s_file,'.xml');
			fb_xml_srv_read.sSymName := '.gst_bestueckbild';
			fb_xml_srv_read.sXPath := '/root/gst_bestueckbild';
			fb_state_entry.i16_next_step := 100;

		ELSIF start_lesen_bestueckbild_halbauto THEN
			s_file := CONCAT(s_path, s_bestueckbild);
			s_file := CONCAT(s_file,'.xml');
			fb_xml_srv_read.sSymName := '.gst_bestueckbild_halbauto';
			fb_xml_srv_read.sXPath := '/root/gst_bestueckbild_halbauto';
			fb_state_entry.i16_next_step := 100;

		ELSIF start_lesen_wkz THEN
			s_file := CONCAT(s_path, s_wkz);
			s_file := CONCAT(s_file,'.xml');
			fb_xml_srv_read.sSymName := '.gst_datensatz.st_wkz';
			fb_xml_srv_read.sXPath := '/root/gst_datensatz.st_wkz';
			fb_state_entry.i16_next_step := 100;
		ELSIF start_lesen_md THEN
			s_file := CONCAT(s_path, s_md);
			s_file := CONCAT(s_file,'.xml');
			fb_xml_srv_read.sSymName := '.gst_datensatz.st_md';
			fb_xml_srv_read.sXPath := '/root/gst_datensatz.st_md';
			fb_state_entry.i16_next_step := 100;
		ELSIF start_lesen_band THEN
			s_file := CONCAT(s_path, s_band);
			s_file := CONCAT(s_file,'.xml');
			fb_xml_srv_read.sSymName := '.gst_datensatz.st_band';
			fb_xml_srv_read.sXPath := '/root/gst_datensatz.st_band';
			fb_state_entry.i16_next_step := 100;
		ELSIF start_lesen_wt THEN
			s_file := CONCAT(s_path, s_wt);
			s_file := CONCAT(s_file,'.xml');
			fb_xml_srv_read.sSymName := '.gst_datensatz.st_wt';
			fb_xml_srv_read.sXPath := '/root/gst_datensatz.st_wt';
			fb_state_entry.i16_next_step := 100;
		END_IF

		(* Daten schreiben *)
		IF start_schreiben_isk THEN
			s_file := CONCAT(s_path, s_isk);
			s_file := CONCAT(s_file,'.xml');
			fb_xml_srv_write.sSymName := '.gst_datensatz.st_isk';
			fb_xml_srv_write.sXPath := '/root/gst_datensatz.st_isk';
			fb_state_entry.i16_next_step := 200;
		ELSIF start_schreiben_bestueckbild THEN
			s_file := CONCAT(s_path, s_bestueckbild);
			s_file := CONCAT(s_file,'.xml');
			fb_xml_srv_write.sSymName := '.gst_bestueckbild';
			fb_xml_srv_write.sXPath := '/root/gst_bestueckbild';
			fb_state_entry.i16_next_step := 200;
		ELSIF start_schreiben_bestueckbild_halbauto THEN
			s_file := CONCAT(s_path, s_bestueckbild);
			s_file := CONCAT(s_file,'.xml');
			fb_xml_srv_write.sSymName := '.gst_bestueckbild_halbauto';
			fb_xml_srv_write.sXPath := '/root/gst_bestueckbild_halbauto';
			fb_state_entry.i16_next_step := 200;
		ELSIF start_schreiben_wkz THEN
			s_file := CONCAT(s_path, s_wkz);
			s_file := CONCAT(s_file,'.xml');
			fb_xml_srv_write.sSymName := '.gst_datensatz.st_wkz';
			fb_xml_srv_write.sXPath := '/root/gst_datensatz.st_wkz';
			fb_state_entry.i16_next_step := 200;
		ELSIF start_schreiben_md_backup THEN
			s_file := CONCAT(s_path, s_md_backup);
			s_file := CONCAT(s_file,'.xml');
			fb_xml_srv_write.sSymName := '.gst_datensatz.st_md';
			fb_xml_srv_write.sXPath := '/root/gst_datensatz.st_md';
			fb_state_entry.i16_next_step := 200;
		ELSIF start_schreiben_md THEN
			s_file := CONCAT(s_path, s_md);
			s_file := CONCAT(s_file,'.xml');
			fb_xml_srv_write.sSymName := '.gst_datensatz.st_md';
			fb_xml_srv_write.sXPath := '/root/gst_datensatz.st_md';
			fb_state_entry.i16_next_step := 200;
		ELSIF start_schreiben_band THEN
			s_file := CONCAT(s_path, s_band);
			s_file := CONCAT(s_file,'.xml');
			fb_xml_srv_write.sSymName := '.gst_datensatz.st_band';
			fb_xml_srv_write.sXPath := '/root/gst_datensatz.st_band';
			fb_state_entry.i16_next_step := 200;
		ELSIF start_schreiben_wt THEN
			s_file := CONCAT(s_path, s_wt);
			s_file := CONCAT(s_file,'.xml');
			fb_xml_srv_write.sSymName := '.gst_datensatz.st_wt';
			fb_xml_srv_write.sXPath := '/root/gst_datensatz.st_wt';
			fb_state_entry.i16_next_step := 200;
		END_IF

(*=======================================================*)
	100:	(* Starte Daten lesen *)
		IF fb_state_entry.E THEN
			fb_xml_srv_read.bExecute := TRUE;
			fb_xml_srv_read.sFilePath := s_file;
		END_IF

		IF fb_xml_srv_read.bBusy THEN
			fb_xml_srv_read.bExecute := FALSE;
			fb_state_entry.i16_next_step := 110;
		END_IF

(*=======================================================*)
	110:	(* Lesevorgang *)
		IF NOT fb_xml_srv_read.bBusy  THEN
			IF NOT fb_xml_srv_read.bError THEN
				fb_state_entry.i16_next_step := 120;
			ELSE	(* Fehler *)
				nErrId := fb_xml_srv_read.nErrId;
				fb_state_entry.i16_next_step := 1000;
			END_IF
		END_IF

(*=======================================================*)
	120:	(* Lesevorgang beendet *)
		IF fb_state_entry.E THEN
			fertig_lesen := TRUE;
		END_IF

		IF 	NOT start_lesen_band AND
			NOT start_lesen_bestueckbild AND
			NOT start_lesen_isk AND
			NOT start_lesen_md AND
			NOT start_lesen_wkz AND
			NOT start_lesen_wt AND
			NOT fb_state_entry.E
			THEN
				fb_state_entry.i16_next_step := 0;
		END_IF

		IF fb_state_entry.X THEN
			fertig_lesen := TRUE;
		END_IF

(*=======================================================*)
	200:	(* Starte Daten schreiben *)
		IF fb_state_entry.E THEN
			fb_xml_srv_write.bExecute := TRUE;
			fb_xml_srv_write.sFilePath := s_file;
		END_IF

		IF fb_xml_srv_write.bBusy THEN
			fb_xml_srv_write.bExecute := FALSE;
			fb_state_entry.i16_next_step := 210;
		END_IF

(*=======================================================*)
	210:	(* Schreibvorgang *)
		IF NOT fb_xml_srv_write.bBusy  THEN
			IF NOT fb_xml_srv_write.bError THEN
				fb_state_entry.i16_next_step := 220;
			ELSE	(* Fehler *)
				nErrId := fb_xml_srv_write.nErrId;
				fb_state_entry.i16_next_step := 1000;
			END_IF
		END_IF

(*=======================================================*)
	220:	(* Schreibvorgang beendet *)
		IF fb_state_entry.E THEN
			fertig_schreiben := TRUE;
		END_IF

		IF 	NOT start_schreiben_band AND
			NOT start_schreiben_bestueckbild AND
			NOT start_schreiben_isk AND
			NOT start_schreiben_md AND
			NOT start_schreiben_md_backup AND
			NOT start_schreiben_wkz AND
			NOT start_schreiben_wt AND
			NOT fb_state_entry.E
			THEN
				fb_state_entry.i16_next_step := 0;
		END_IF

		IF fb_state_entry.X THEN
			fertig_schreiben := TRUE;
		END_IF

(*=======================================================*)
	1000: (* Fehler *)
		IF fb_state_entry.E THEN
			bError := TRUE;
			fb_ton_quitt.IN := FALSE;
		END_IF

		(*-----------------------Weiterschaltbedingungen----------------------------*)
		IF bQuit AND NOT fb_state_entry.E THEN
			bError := FALSE;
			fb_ton_quitt.IN := TRUE;
		END_IF

		IF fb_ton_quitt.Q THEN
			fb_ton_quitt.IN := FALSE;
			fb_state_entry.i16_next_step := 0;
		END_IF
END_CASE


fb_state_entry(
	i16_next_step:= ,
	i16_pos:= 2,
	s_debugtext:= ,
	E=> ,
	X=> ,
	i16_step=> ,
	i16_last_step=> );

(* XML *)
fb_xml_srv_read(
	sNetId:= '',
	ePath:= PATH_GENERIC,
	nMode:= XMLSRV_SKIPMISSING,
	sSymName:= ,
	sFilePath:= ,
	sXPath:= ,
	bExecute:= ,
	tTimeout:= t#10s,
	bBusy=> ,
	bError=> ,
	nErrId=> );

fb_xml_srv_write(
	sNetId:= '',
	ePath:= PATH_GENERIC,
	nMode:= XMLSRV_ADDMISSING,
	sSymName:=  ,
	sFilePath:= ,
	sXPath:= ,
	bExecute:= ,
	tTimeout:= t#10s,
	bBusy=> ,
	bError=> ,
	nErrId=> );
END_FUNCTION_BLOCK

(* POU Gemeinsamkeiten17xx/BBGen/ST_BBGenWriteFile, ST *)
FUNCTION_BLOCK ST_BBGenWriteFile
VAR_INPUT
	bStart		: BOOL;
END_VAR
VAR_OUTPUT
	bFertig	: BOOL;
	bError	: BOOL;
END_VAR
VAR
	fb_state_entry						: ST_StateEntry;
	fb_r_trig_start						: R_TRIG;
	fb_ton_quitt						: TON;
	fb_openfile						: FILEOPEN;
	fb_writefile						: FILEWRITE;
	fb_closefile						: FILECLOSE;

	s_file							: STRING(255);

	nErrId							: DINT;

	tmp								: DINT;
	lo								: DINT;
	ll								: DINT;
	s_line							: STRING(255);
	s_out							: STRING(10000);
	y								: STRING;
	z								: STRING;
	b								: STRING;
	tab								: STRING;
	lineend							: STRING;
END_VAR
fb_ton_quitt(IN:= , PT:= t#50ms, Q=> , ET=> );
fb_r_trig_start(CLK:= bStart, Q=> );
(* ======================================Schrittkette======================================== *)
fb_state_entry(
	i16_next_step:= ,
	i16_pos:= 1,
	s_debugtext:= ,
	E=> ,
	X=> ,
	i16_step=> ,
	i16_last_step=> );


CASE fb_state_entry.i16_step OF
(*=======================================================*)
	0:
		nErrId := 0;

		bFertig := FALSE;
		bError := FALSE;

		s_file := 'D:\BBGen\bbgen.txt';
		fb_state_entry.i16_next_step := 10;
(*=======================================================*)
	10:
		IF fb_r_trig_start.Q THEN
			fb_state_entry.i16_next_step := 100;
		END_IF
(*=======================================================*)
	100:
		(* Öffne Datei *)
		IF fb_state_entry.E THEN
			fb_openfile.OPEN := TRUE;
		END_IF

		IF fb_openfile.ERR THEN
			fb_state_entry.i16_next_step := FEHLER;
			nErrId := fb_openfile.ERRID;
		END_IF

		IF NOT fb_state_entry.E AND NOT fb_openfile.BUSY AND NOT fb_openfile.ERR THEN
			fb_state_entry.i16_next_step := 110;
		END_IF

		IF fb_state_entry.X THEN
			fb_openfile.OPEN := FALSE;
		END_IF
(*=======================================================*)
	110:
		(* Datei ist offen. Schreibe Einträge*)
		IF fb_state_entry.E THEN
			(* Baue Ausgabestring *)
			s_out := '';
			tab := '$T';
			lineend := '$R$N';
			lo := 0;
			ll := 0;
			(* Erste Zeile: Offset und Breite/Höhe*)
			y := LREAL_TO_FMTSTR(gst_datensatz.st_isk.lr_pos_y_0,2,TRUE);	s_line := CONCAT(y,tab);
			z := LREAL_TO_FMTSTR(gst_datensatz.st_isk.lr_pos_z_0,2,TRUE);	s_line := CONCAT(s_line,z);	s_line := CONCAT(s_line,tab);

			y := LREAL_TO_FMTSTR(gst_datensatz.st_isk.lr_breite,2,TRUE);		s_line := CONCAT(s_line,y);	s_line := CONCAT(s_line,tab);
			z := LREAL_TO_FMTSTR(gst_datensatz.st_isk.lr_hoehe,2,TRUE);		s_line := CONCAT(s_line,z);	s_line := CONCAT(s_line,lineend);
			s_out := s_line; lo := LEN(s_out);

			FOR tmp := 0 TO gst_datensatz.st_bestueckprogramm.i32_anzahl-1 BY 1
			DO
				y := LREAL_TO_FMTSTR (gst_datensatz.st_bestueckprogramm.lr_y[tmp],2,TRUE);
				z := LREAL_TO_FMTSTR(gst_datensatz.st_bestueckprogramm.lr_z[tmp],2,TRUE);
				b := INT_TO_STRING(gst_datensatz.st_bestueckprogramm.i16_b[tmp]);
				s_line := y;						ll := LEN(y);
				s_line := CONCAT(s_line, tab);		ll := ll + LEN(tab);
				s_line := CONCAT(s_line, z);			ll := ll + LEN(z);
				s_line := CONCAT(s_line, tab);		ll := ll + LEN(tab);
				s_line := CONCAT(s_line, b);			ll := ll + LEN(b);
				s_line := CONCAT(s_line, lineend);	ll := ll + LEN(lineend);

				(* Da concat und co nur Strings bis 255 Zeichen kann, müssen wir hier memcpy nutzen *)
				MEMCPY(ADR(s_out)+lo,ADR(s_line), ll);
				lo := lo + ll;
			END_FOR
			fb_writefile.BUFADDR := ADR(s_out);
			fb_writefile.COUNT := lo;
			fb_writefile.WRITE := TRUE;
		END_IF

		IF NOT fb_state_entry.E AND fb_writefile.ERR  THEN
			fb_state_entry.i16_next_step := FEHLER;
			nErrId := fb_writefile.ERRID;
		END_IF

		IF NOT fb_state_entry.E AND NOT fb_writefile.BUSY AND NOT fb_writefile.ERR THEN
			(* Erfolgreich geschrieben *)
			fb_state_entry.i16_next_step := 200;
		END_IF

		IF fb_state_entry.X THEN
			fb_writefile.WRITE := FALSE;
		END_IF

(*=======================================================*)
	200:
		(* Schliesse Datei *)
		IF fb_state_entry.E THEN
			fb_closefile.CLOSE := TRUE;
		END_IF

		IF fb_closefile.ERR THEN
			fb_state_entry.i16_next_step := FEHLER;
			nErrId := fb_closefile.ERRID;
		END_IF

		IF NOT fb_state_entry.E AND NOT fb_closefile.BUSY AND NOT fb_closefile.ERR THEN
			fb_state_entry.i16_next_step := 210;
		END_IF

		IF fb_state_entry.X THEN
			fb_closefile.CLOSE := FALSE;
		END_IF

(*=======================================================*)
	210:
		IF fb_state_entry.E THEN
			bFertig := TRUE;
		END_IF

		IF NOT bStart AND NOT fb_state_entry.E THEN
			fb_state_entry.i16_next_step := 10;
		END_IF

		IF fb_state_entry.X THEN
			bFertig := FALSE;
		END_IF

(*=======================================================*)
	1000: (* Fehler *)
		IF fb_state_entry.E THEN
			bError := TRUE;
			fb_ton_quitt.IN := FALSE;
		END_IF

		(*-----------------------Weiterschaltbedingungen----------------------------*)
		IF NOT fb_state_entry.E THEN
			bError := FALSE;
			fb_ton_quitt.IN := TRUE;
		END_IF

		IF fb_ton_quitt.Q THEN
			fb_ton_quitt.IN := FALSE;
			fb_state_entry.i16_next_step := 0;
		END_IF
END_CASE

fb_state_entry(
	i16_next_step:= ,
	i16_pos:= 2,
	s_debugtext:= ,
	E=> , 
	X=> ,
	i16_step=> ,
	i16_last_step=> );

(* FILE *)
fb_openfile(
	NETID:= ,
	FPATHNAME:= s_file,
	OPENMODE:= FILE_OPENWRITE, (* Wir wollen eine bestehenede Datei im Falle überschreiben *)
	OPEN:= ,
	TMOUT:= t#2s,
	BUSY=> , 
	ERR=> , 
	ERRID=> , 
	HFILE=> );

fb_writefile(
	NETID:= ,
	HFILE:= fb_openfile.HFILE,
	BUFADDR:= , 
	COUNT:= ,
	WRITE:= ,
	TMOUT:= t#2s,
	BUSY=> ,
	ERR=> ,
	ERRID=> ,
	COUNT_W=> );

fb_closefile(
	NETID:= , 
	HFILE:= fb_openfile.HFILE,
	CLOSE:= , 
	TMOUT:= t#2s,
	BUSY=> ,
	ERR=> , 
	ERRID=> );
END_FUNCTION_BLOCK

(* POU EPT Lib/Funktionsbausteine/ST_Export_String, ST *)
FUNCTION_BLOCK ST_Export_String
VAR_INPUT
	Start				:BOOL;
	ExportStr			:STRING(255);
	FileName			:STRING;
	Path				:STRING;
	Mode				:DWORD;
END_VAR
VAR
	fb_state_entry		:ST_StateEntry;
	fb_file_open			:FB_FileOpen;
	fb_file_puts			:FB_FilePuts;
	fb_file_close			:FB_FileClose;
	nErrId					:UDINT;
	ErrorMsg			:STRING(255);
	hFile				:UINT;
END_VAR
VAR_OUTPUT
	Ready				:BOOL;
	Busy				:BOOL;
	Done				:BOOL;
	Error				:BOOL;
END_VAR
fb_state_entry(i16_pos:= 1);

CASE fb_state_entry.i16_step OF

(*=======================================================*)
	0:	(*Objekt initialisieren*)

		(*-----------------------Weiterschaltbedingungen----------------------------*)
		fb_state_entry.i16_next_step:=INIT;

(*=======================================================*)
	10:	(*initialisieren*)

		(*-----------------------Weiterschaltbedingungen----------------------------*)
		fb_state_entry.i16_next_step:=BEREIT;

(*=======================================================*)
	BEREIT:(*Start*)

		(*-----------------------Weiterschaltbedingungen----------------------------*)
		IF Start THEN
			Start:=FALSE;
			Busy:=TRUE;
			Error:=FALSE;
			Done:=FALSE;
			nErrId:=0;
			ErrorMsg:='';
			fb_state_entry.i16_next_step:=105;
		END_IF

(*=======================================================*)
	105: (*Datei erstellen*)
		IF fb_state_entry.E THEN
			fb_file_open.sPathName:=CONCAT (Path, FileName);
			fb_file_open.bExecute:=TRUE;
		END_IF

		(*-----------------------Weiterschaltbedingungen----------------------------*)
		IF  fb_file_open.bBusy THEN
			fb_state_entry.i16_next_step:=110;
		END_IF

(*=======================================================*)
	110: (*Datei erstellen*)

		(*-----------------------Weiterschaltbedingungen----------------------------*)
		IF 	NOT fb_file_open.bBusy THEN
			fb_file_open.bExecute:=FALSE;
			IF 	fb_file_open.bError THEN
				nErrId:=fb_file_open.nErrId;
				fb_state_entry.i16_next_step:=FEHLER;
				ErrorMsg:='Fehler beim Öffnen der Datei';
			ELSE
				fb_state_entry.i16_next_step:=120;
			END_IF
		END_IF

(*=======================================================*)
	120: (*String in Datei eintragen*)
		IF fb_state_entry.E THEN
			fb_file_puts.sLine:=ExportStr;
			fb_file_puts.bExecute:=TRUE;
		END_IF

		(*-----------------------Weiterschaltbedingungen----------------------------*)
		IF  fb_file_puts.bBusy THEN
			fb_state_entry.i16_next_step:=130;
		END_IF

(*=======================================================*)
	130: (*String in Datei eintragen*)

		(*-----------------------Weiterschaltbedingungen----------------------------*)
		IF 	NOT fb_file_puts.bBusy THEN
			fb_file_puts.bExecute:=FALSE;
			IF 	fb_file_puts.bError THEN
				nErrId:=fb_file_puts.nErrId;
				fb_state_entry.i16_next_step:=FEHLER;
			ELSE
				fb_state_entry.i16_next_step:=140;
			END_IF
		END_IF
	
(*=======================================================*)
	140:(*Datei schließen*)
		IF fb_state_entry.E THEN
		fb_file_close.bExecute:=TRUE;
		END_IF

		(*-----------------------Weiterschaltbedingungen----------------------------*)
		IF 	fb_file_close.bBusy THEN
			fb_state_entry.i16_next_step:=150;
		END_IF
	
(*=======================================================*)
	150:(*Datei schließen*)

		(*-----------------------Weiterschaltbedingungen----------------------------*)
		IF NOT fb_file_close.bBusy THEN
			fb_file_close.bExecute:=FALSE;
			IF 	fb_file_close.bError THEN
				nErrId:=fb_file_close.nErrId;
				fb_state_entry.i16_next_step:=FEHLER;
				ErrorMsg:='Fehler beim Schließen der Datei';
			ELSE
				Busy:=FALSE;
				Done:=TRUE;
				fb_state_entry.i16_next_step:=BEREIT;
			END_IF
		END_IF

(*=======================================================*)
	FEHLER:	(*bei Fehler einfach weiter*)

		Busy:=FALSE;
		Error:=TRUE;
		fb_state_entry.i16_next_step := INIT;

END_CASE

fb_state_entry(i16_pos:= 2);


fb_file_open(
	sNetId:='',
	sPathName:= ,
	nMode:=Mode,
	ePath:=PATH_GENERIC,
	bExecute:= ,
	tTimeout:=T#1s,
	hFile=> hFile);

fb_file_puts(
	sNetId:='',
	hFile:=hFile,
	sLine:= ,
	bExecute:= ,
	tTimeout:=t#1s);

fb_file_close(
	sNetId:='',
	hFile:=hFile,
	bExecute:= ,
	tTimeout:=t#1s);
END_FUNCTION_BLOCK

(* POU Gemeinsamkeiten17xx/Safety/ST_Safetyprogramm, ST *)
PROGRAM ST_Safetyprogramm
VAR_INPUT
	st_config							: struct_config;
	st_ctrl_in							: struct_ctrl_in;
END_VAR
VAR_IN_OUT
	st_visu							: struct_visu;
END_VAR
VAR_OUTPUT
	st_ctrl_out						: struct_ctrl_out;
END_VAR
VAR
	ack_step							: ST_StateEntry;
	fb_ton_wz						: TON;
	fb_ton_quitt						: TON;
	fb_ton_taste_steuerung_ein				: TON;
	fb_ton_taste_steuerung_aus				: TON;
	fb_ton_taste_stoerung_quitt				: TON;
	fb_r_trig_quittieren					: R_TRIG;
	fb_state_entry						: ST_StateEntry;
	i32_fb_error_counter_gruppe1		: DINT := 0;
	i32_fb_error_counter_gruppe2		: DINT := 0;
	i32_fb_error_counter_gruppe3		: DINT := 0;
	i32_fb_error_counter_gruppe4		: DINT := 0;
	i32_com_error_counter_gruppe1		: DINT := 0;
	i32_com_error_counter_gruppe2		: DINT := 0;
	i32_com_error_counter_gruppe3		: DINT := 0;
	i32_com_error_counter_gruppe4		: DINT := 0;

	sm_steuerung_aus				: BOOL := FALSE;
	sm_not_halt_intern					: BOOL := FALSE;
	sm_not_halt_frontseite				: BOOL := FALSE;
	sm_not_halt_rueckseite			: BOOL := FALSE;
	sm_not_halt_bediengeraet			: BOOL := FALSE;
	sm_not_halt_extern				: BOOL := FALSE;
	sm_tuere_vorne_offen				: BOOL := FALSE;
	sm_tuere_hinten_offen				: BOOL := FALSE;
	sm_tuere_vorne_diskrepanz		: BOOL := FALSE;
	sm_tuere_hinten_diskrepanz		: BOOL := FALSE;
	sm_bestueckachse_sto			: BOOL := FALSE;
	sm_bestueckachse_sls			: BOOL := FALSE;
	sm_z_achse_sto					: BOOL := FALSE;
	sm_z_achse_sls					: BOOL := FALSE;
	sm_y_achse_sto					: BOOL := FALSE;
	sm_y_achse_sls					: BOOL := FALSE;
	sm_b_achse_sto					: BOOL := FALSE;
	sm_b_achse_sls					: BOOL := FALSE;
	sm_transport_achse_sto				: BOOL := FALSE;
	sm_transport_achse_sls			: BOOL := FALSE;

	bm_taste_steuerung_ein_verhaengt		: BOOL := FALSE;
	bm_taste_steuerung_aus_verhaengt		: BOOL := FALSE;
	bm_taste_stoerung_quitt_verhaengt		: BOOL := FALSE;

	sm_fehler_fb1_opmode					: BOOL := FALSE;
	sm_fehler_fb9_estop_nothalt_front			: BOOL := FALSE;
	sm_fehler_fb10_estop_nothalt_ext			: BOOL := FALSE;
	sm_fehler_fb15_edm_nothalt_ext				: BOOL := FALSE;
	sm_fehler_fb16_edm_nothalt_schuetz			: BOOL := FALSE;
	sm_fehler_fb17_edm_ventilinsel				: BOOL := FALSE;
	sm_fehler_fb28_edm_foerderband			: BOOL := FALSE;
	sm_fehler_fb30_estop_rueck				: BOOL := FALSE;
	sm_fehler_fb31_estop_bedien				: BOOL := FALSE;
	sm_fehler_fb35_mon_tuere_vo				: BOOL := FALSE;
	sm_fehler_fb36_mon_tuere_hi				: BOOL := FALSE;
	sm_fehler_fb37_mon_tuere_disk_vo			: BOOL := FALSE;
	sm_fehler_fb38_mon_tuere_disk_hi			: BOOL := FALSE;
	sm_fehler_fb39_mon_tuere_meld_vo			: BOOL := FALSE;
	sm_fehler_fb40_mon_tuere_meld_hi			: BOOL := FALSE;
	sm_not_halt_hublift_links					: BOOL := FALSE;

	a_quitt_pilz_hublift_links			AT %Q* : BOOL;

	a_lampe_quitt_schutztuere_vorne	AT %Q* : BOOL;
	a_lampe_quitt_schutztuere_hinten	AT %Q* : BOOL;

	(* Eingänge von Twinsafe FBs *)
	se_quittiertaste					AT %I* : BOOL;
	se_taste_steuerung_ein				AT %I* : BOOL;
	se_taste_steuerung_aus				AT %I* : BOOL;
	se_steuerung_ein					AT %I* : BOOL;
	se_ba_mit_bedingungen				AT %I* : BOOL;
	se_nothalt_gesamt_ok				AT %I* : BOOL;
	se_tuere_vorne_diskrepanz			AT %I* : BOOL;
	se_tuere_hinten_diskrepanz			AT %I* : BOOL;
	se_not_halt_intern					AT %I* : BOOL;
	se_not_halt_frontseite				AT %I* : BOOL;
	se_not_halt_rueckseite				AT %I* : BOOL;
	se_not_halt_bediengeraet			AT %I* : BOOL;
	se_not_halt_extern					AT %I* : BOOL;
	se_tuere_vorne_offen				AT %I* : BOOL;
	se_tuere_hinten_offen				AT %I* : BOOL;
	se_tuere_zustimm_vorne_offen		AT %I* : BOOL;
	se_tuere_zustimm_hinten_offen		AT %I* : BOOL;
	se_bestueckachse_sto				AT %I* : BOOL;
	se_bestueckachse_sls				AT %I* : BOOL;
	se_z_achse_sto					AT %I* : BOOL;
	se_z_achse_sls					AT %I* : BOOL;
	se_y_achse_sto					AT %I* : BOOL;
	se_y_achse_sls					AT %I* : BOOL;
	se_b_achse_sto					AT %I* : BOOL;
	se_b_achse_sls					AT %I* : BOOL;
	se_transport_achse_sto			AT %I* : BOOL;
	se_transport_achse_sls			AT %I* : BOOL;

	e_not_halt_hublift_links_ok				AT %I* : BOOL;	(* Not Halt OK Signal von Pilz Hublift links *)

	se_fehler_fb1_opmode						AT %I* : BOOL;
	se_fehler_fb9_estop_nothalt_front			AT %I* : BOOL;
	se_fehler_fb10_estop_nothalt_ext			AT %I* : BOOL;
	se_fehler_fb15_edm_nothalt_ext				AT %I* : BOOL;
	se_fehler_fb16_edm_nothalt_schuetz			AT %I* : BOOL;
	se_fehler_fb17_edm_ventilinsel				AT %I* : BOOL;
	se_fehler_fb28_edm_foerderband			AT %I* : BOOL;
	se_fehler_fb30_estop_rueck				AT %I* : BOOL;
	se_fehler_fb31_estop_bedien				AT %I* : BOOL;
	se_fehler_fb35_mon_tuere_vo				AT %I* : BOOL;
	se_fehler_fb36_mon_tuere_hi				AT %I* : BOOL;
	se_fehler_fb37_mon_tuere_disk_vo			AT %I* : BOOL;
	se_fehler_fb38_mon_tuere_disk_hi			AT %I* : BOOL;
	se_fehler_fb39_mon_tuere_meld_vo			AT %I* : BOOL;
	se_fehler_fb40_mon_tuere_meld_hi			AT %I* : BOOL;

	(* Betriebsarten *)
	sa_run_stop_gruppe1				AT %Q* : BOOL;
	sa_err_ack_gruppe1				AT %Q* : BOOL;
	se_fb_error_gruppe1				AT %I* : BOOL;
	se_com_error_gruppe1			AT %I* : BOOL;
	se_out_error_gruppe1				AT %I* : BOOL;
	(* Notaus *)
	sa_run_stop_gruppe2				AT %Q* : BOOL;
	sa_err_ack_gruppe2				AT %Q* : BOOL;
	se_fb_error_gruppe2				AT %I* : BOOL;
	se_com_error_gruppe2			AT %I* : BOOL;
	se_out_error_gruppe2				AT %I* : BOOL;
	(* Türen *)
	sa_run_stop_gruppe3				AT %Q* : BOOL;
	sa_err_ack_gruppe3				AT %Q* : BOOL;
	se_fb_error_gruppe3				AT %I* : BOOL;
	se_com_error_gruppe3			AT %I* : BOOL;
	se_out_error_gruppe3				AT %I* : BOOL;
	(* Safety AX5000 *)
	sa_run_stop_gruppe4				AT %Q* : BOOL;
	sa_err_ack_gruppe4				AT %Q* : BOOL;
	se_fb_error_gruppe4				AT %I* : BOOL;
	se_com_error_gruppe4			AT %I* : BOOL;
	se_out_error_gruppe4				AT %I* : BOOL;
END_VAR
(* Zeiten *)
fb_ton_wz(IN:= , PT:= T#100ms, Q=>  , ET=> );
fb_ton_quitt(IN:= , PT:= t#20ms, Q=> , ET=> );
fb_ton_taste_steuerung_ein(IN:= se_taste_steuerung_ein, PT:= t#60s, Q=> bm_taste_steuerung_ein_verhaengt, ET=> );
fb_ton_taste_steuerung_aus(IN:= NOT se_taste_steuerung_aus, PT:= t#60s, Q=> bm_taste_steuerung_aus_verhaengt, ET=> );
fb_ton_taste_stoerung_quitt(IN:= se_quittiertaste, PT:= t#60s, Q=> bm_taste_stoerung_quitt_verhaengt, ET=> );

(* Flanken *)
fb_r_trig_quittieren(CLK:= visu.b_quittieren, Q=> );

(* Startsignal für die Safety-Gruppen *)
sa_run_stop_gruppe1 := TRUE;
sa_run_stop_gruppe2 := TRUE;
sa_run_stop_gruppe3 := TRUE;
sa_run_stop_gruppe4 := TRUE;

(* Automatische Quittierung von Errors in den TwinSafe-Gruppen *)
ack_step(
	i16_next_step:= ,
	i16_pos:= 1,
	s_debugtext:= ,
	E=> ,
	X=> ,
	i16_step=> ,
	i16_last_step=> );

CASE ack_step.i16_step OF
	0:	(* Nach Startup automatische Quittierung von FB- und COM-Fehlern *)
		IF 	se_fb_error_gruppe1 OR
			se_com_error_gruppe1 OR
			se_fb_error_gruppe2 OR
			se_com_error_gruppe2 OR
			se_fb_error_gruppe3 OR
			se_com_error_gruppe3 OR
			se_fb_error_gruppe4 OR
			se_com_error_gruppe4
			THEN
				sa_err_ack_gruppe1 := FALSE;
				sa_err_ack_gruppe2 := FALSE;
				sa_err_ack_gruppe3 := FALSE;
				sa_err_ack_gruppe4 := FALSE;
				fb_ton_wz.IN := TRUE;
				IF fb_ton_wz.Q THEN
					fb_ton_wz.IN := FALSE;
					ack_step.i16_next_step := 10;
				END_IF
		END_IF

	10:
		sa_err_ack_gruppe1 := TRUE;
		sa_err_ack_gruppe2 := TRUE;
		sa_err_ack_gruppe3 := TRUE;
		sa_err_ack_gruppe4 := TRUE;
		fb_ton_wz.IN := TRUE;
		IF fb_ton_wz.Q THEN
			fb_ton_wz.IN := FALSE;
			ack_step.i16_next_step := 20;
		END_IF

	20:
		sa_err_ack_gruppe1 := FALSE;
		sa_err_ack_gruppe2 := FALSE;
		sa_err_ack_gruppe3 := FALSE;
		sa_err_ack_gruppe4 := FALSE;
		fb_ton_wz.IN := TRUE;
		IF fb_ton_wz.Q THEN
			fb_ton_wz.IN := FALSE;
			ack_step.i16_next_step := 100;
		END_IF

	100:	(* FB- und COM-Fehler  *)
		IF 	se_fb_error_gruppe1 OR
			se_com_error_gruppe1 OR
			se_fb_error_gruppe2 OR
			se_com_error_gruppe2 OR
			se_fb_error_gruppe3 OR
			se_com_error_gruppe3 OR
			se_fb_error_gruppe4 OR
			se_com_error_gruppe4
			THEN
				sa_err_ack_gruppe1 := FALSE;
				sa_err_ack_gruppe2 := FALSE;
				sa_err_ack_gruppe3 := FALSE;
				sa_err_ack_gruppe4 := FALSE;
				ack_step.i16_next_step := 110;
		END_IF

	110:
		IF ack_step.E THEN
			IF se_fb_error_gruppe1 THEN
				i32_fb_error_counter_gruppe1 := i32_fb_error_counter_gruppe1 + 1;
			END_IF
			IF se_fb_error_gruppe2 THEN
				i32_fb_error_counter_gruppe2 := i32_fb_error_counter_gruppe2 + 1;
			END_IF
			IF se_fb_error_gruppe3 THEN
				i32_fb_error_counter_gruppe3 := i32_fb_error_counter_gruppe3 + 1;
			END_IF
			IF se_fb_error_gruppe4 THEN
				i32_fb_error_counter_gruppe4 := i32_fb_error_counter_gruppe4 + 1;
			END_IF
			IF se_com_error_gruppe1 THEN
				i32_com_error_counter_gruppe1 := i32_com_error_counter_gruppe1 + 1;
			END_IF
			IF se_com_error_gruppe2 THEN
				i32_com_error_counter_gruppe2 := i32_com_error_counter_gruppe2 + 1;
			END_IF
			IF se_com_error_gruppe3 THEN
				i32_com_error_counter_gruppe3 := i32_com_error_counter_gruppe3 + 1;
			END_IF
			IF se_com_error_gruppe4 THEN
				i32_com_error_counter_gruppe4 := i32_com_error_counter_gruppe4 + 1;
			END_IF
		END_IF
		ack_step.i16_next_step := 120;

	120:
		sa_err_ack_gruppe1 := TRUE;
		sa_err_ack_gruppe2 := TRUE;
		sa_err_ack_gruppe3 := TRUE;
		sa_err_ack_gruppe4 := TRUE;
		fb_ton_wz.IN := TRUE;
		IF fb_ton_wz.Q THEN
			fb_ton_wz.IN := FALSE;
			ack_step.i16_next_step := 130;
		END_IF

	130:
		sa_err_ack_gruppe1 := FALSE;
		sa_err_ack_gruppe2 := FALSE;
		sa_err_ack_gruppe3 := FALSE;
		sa_err_ack_gruppe4 := FALSE;
		fb_ton_wz.IN := TRUE;
		IF fb_ton_wz.Q THEN
			fb_ton_wz.IN := FALSE;
			ack_step.i16_next_step := 100;
		END_IF
END_CASE

ack_step(
	i16_next_step:= ,
	i16_pos:= 2,
	s_debugtext:= ,
	E=> ,
	X=> , 
	i16_step=> ,
	i16_last_step=> );


(* Lampen für Schutztüren *)
a_lampe_quitt_schutztuere_hinten := NOT se_tuere_hinten_offen;
a_lampe_quitt_schutztuere_vorne := 	NOT se_tuere_vorne_offen OR
								NOT se_tuere_hinten_offen OR
								NOT se_not_halt_intern;

(* Quittierung Pilz Hublift links *)
a_quitt_pilz_hublift_links := se_quittiertaste;

(* ======================================Schrittkette======================================== *)
fb_state_entry(
	i16_next_step:= ,
	i16_pos:= 1,
	s_debugtext:= ,
	E=> ,
	X=> ,
	i16_step=> ,
	i16_last_step=> );

CASE fb_state_entry.i16_step OF
(*=======================================================*)
	INIT_OBJ:
		IF	st_config.b_config_fertig AND
			NOT se_fb_error_gruppe1 AND
			NOT se_com_error_gruppe1 AND
			NOT se_fb_error_gruppe2 AND
			NOT se_com_error_gruppe2 AND
			NOT se_fb_error_gruppe3 AND
			NOT se_com_error_gruppe3 AND
			NOT se_fb_error_gruppe4 AND
			NOT se_com_error_gruppe4
			THEN
				fb_state_entry.i16_next_step := INIT;
		END_IF

(*=======================================================*)
	INIT:
		st_ctrl_out.b_fehler := FALSE;
		st_ctrl_out.b_bereit := FALSE;
		fb_ton_quitt.IN := FALSE;
		sm_steuerung_aus := FALSE;
		sm_not_halt_intern := FALSE;
		sm_not_halt_frontseite := FALSE;
		sm_not_halt_rueckseite := FALSE;
		sm_not_halt_bediengeraet := FALSE;
		sm_not_halt_extern := FALSE;
		sm_tuere_vorne_offen := FALSE;
		sm_tuere_hinten_offen := FALSE;
		sm_tuere_vorne_diskrepanz := FALSE;
		sm_tuere_hinten_diskrepanz := FALSE;
		sm_bestueckachse_sto := FALSE;
		sm_bestueckachse_sls := FALSE;
		sm_z_achse_sto := FALSE;
		sm_z_achse_sls := FALSE;
		sm_y_achse_sto := FALSE;
		sm_y_achse_sls := FALSE;
		sm_b_achse_sto := FALSE;
		sm_b_achse_sls := FALSE;
		sm_transport_achse_sto := FALSE;
		sm_transport_achse_sls := FALSE;
		sm_fehler_fb1_opmode := FALSE;
		sm_fehler_fb9_estop_nothalt_front := FALSE;
		sm_fehler_fb10_estop_nothalt_ext := FALSE;
		sm_fehler_fb15_edm_nothalt_ext	 := FALSE;
		sm_fehler_fb16_edm_nothalt_schuetz := FALSE;
		sm_fehler_fb17_edm_ventilinsel := FALSE;
		sm_fehler_fb28_edm_foerderband := FALSE;
		sm_fehler_fb30_estop_rueck := FALSE;
		sm_fehler_fb31_estop_bedien := FALSE;
		sm_fehler_fb35_mon_tuere_vo := FALSE;
		sm_fehler_fb36_mon_tuere_hi := FALSE;
		sm_fehler_fb37_mon_tuere_disk_vo := FALSE;
		sm_fehler_fb38_mon_tuere_disk_hi := FALSE;
		sm_fehler_fb39_mon_tuere_meld_vo := FALSE;
		sm_fehler_fb40_mon_tuere_meld_hi := FALSE;
		sm_not_halt_hublift_links := FALSE;

		(*-----------------------Weiterschaltbedingungen----------------------------*)
		fb_state_entry.i16_next_step := BEREIT;

(*=======================================================*)
	BEREIT:
		IF fb_state_entry.E THEN
			st_ctrl_out.b_bereit := TRUE;
		END_IF

		(* Hinweis: SLS der Achsen endet immer bei STO, deshalb wird nur STO abgefragt *)
		CASE gst_datensatz.st_md.i16_typ_zelle OF
			KEINE_ZELLE:
				;

			BESTUECKZELLE_1700, RASTERFOLIE:
				IF	se_steuerung_ein AND
					se_not_halt_intern AND
					se_not_halt_extern AND
					se_tuere_zustimm_vorne_offen AND
					se_tuere_zustimm_hinten_offen AND
					(*se_tuere_vorne_offen AND
					se_tuere_hinten_offen AND*)
					NOT se_bestueckachse_sto AND
					NOT se_z_achse_sto AND
					NOT se_y_achse_sto AND
					NOT se_tuere_vorne_diskrepanz AND
					NOT se_tuere_hinten_diskrepanz AND
					(e_not_halt_hublift_links_ok OR NOT gst_datensatz.st_md.b_hublift_links_aktiv)
					THEN
						;
				ELSE
					fb_state_entry.i16_next_step := FEHLER;
				END_IF

			BESTUECKZELLE_1720:
				IF	se_steuerung_ein AND
					se_not_halt_intern AND
					se_not_halt_extern AND
					se_tuere_zustimm_vorne_offen AND
					se_tuere_zustimm_hinten_offen AND
					(*se_tuere_vorne_offen AND
					se_tuere_hinten_offen AND*)
					NOT se_bestueckachse_sto AND
					NOT se_z_achse_sto AND
					NOT se_tuere_vorne_diskrepanz AND
					NOT se_tuere_hinten_diskrepanz AND
					(e_not_halt_hublift_links_ok OR NOT gst_datensatz.st_md.b_hublift_links_aktiv)
					THEN
						;
				ELSE
					fb_state_entry.i16_next_step := FEHLER;
				END_IF
		END_CASE

(*=======================================================*)
	FEHLER:
		IF fb_state_entry.E THEN
			st_ctrl_out.b_fehler := TRUE;
			fb_ton_quitt.IN := FALSE;
		END_IF

		(* Gruppe NOT-AUS *)
		sm_not_halt_frontseite := NOT se_not_halt_frontseite;
		sm_not_halt_rueckseite := NOT se_not_halt_rueckseite;
		sm_not_halt_bediengeraet := NOT se_not_halt_bediengeraet;
		sm_steuerung_aus := NOT se_steuerung_ein AND se_not_halt_frontseite AND se_not_halt_rueckseite AND se_not_halt_bediengeraet AND se_tuere_vorne_offen AND se_tuere_hinten_offen;
		sm_not_halt_extern := NOT se_not_halt_extern;

		IF se_steuerung_ein AND se_not_halt_frontseite AND se_not_halt_rueckseite AND se_not_halt_bediengeraet THEN
			(* Gruppe Achsen *)
			sm_bestueckachse_sto := 	se_bestueckachse_sto AND
									(gst_datensatz.st_md.i16_typ_zelle = BESTUECKZELLE_1700 OR gst_datensatz.st_md.i16_typ_zelle = BESTUECKZELLE_1720);
			sm_z_achse_sto := se_z_achse_sto;
			sm_y_achse_sto := se_y_achse_sto AND
								gst_datensatz.st_md.i16_typ_zelle = BESTUECKZELLE_1700 ;
			sm_b_achse_sto := se_b_achse_sto AND
							(gst_datensatz.st_wkz.i16_typ_bandeinzug = SERVO);
			sm_transport_achse_sto := se_transport_achse_sto AND
							(gst_datensatz.st_md.b_anwahl_transport_achse);
		END_IF

		(* Gruppe Schutzeinrichtungen *)
		(* Schutztüren Bestückautomat vorne *)
		sm_tuere_vorne_offen :=  NOT se_tuere_vorne_offen;
		sm_tuere_vorne_diskrepanz := se_tuere_vorne_diskrepanz;
		(* Schutztüren Bestückautomat hinten *)
		sm_tuere_hinten_offen := NOT se_tuere_hinten_offen;
		sm_tuere_hinten_diskrepanz := se_tuere_hinten_diskrepanz;

		(* SAFETY- FB-Fehler *)
		sm_fehler_fb1_opmode := se_fehler_fb1_opmode;
		sm_fehler_fb9_estop_nothalt_front := se_fehler_fb9_estop_nothalt_front;
		sm_fehler_fb10_estop_nothalt_ext := se_fehler_fb10_estop_nothalt_ext;
		sm_fehler_fb15_edm_nothalt_ext := se_fehler_fb15_edm_nothalt_ext;
		sm_fehler_fb16_edm_nothalt_schuetz := se_fehler_fb16_edm_nothalt_schuetz;
		sm_fehler_fb17_edm_ventilinsel := se_fehler_fb17_edm_ventilinsel;
		sm_fehler_fb28_edm_foerderband := se_fehler_fb28_edm_foerderband;
		sm_fehler_fb30_estop_rueck := se_fehler_fb30_estop_rueck;
		sm_fehler_fb31_estop_bedien := se_fehler_fb31_estop_bedien;
		sm_fehler_fb35_mon_tuere_vo := se_fehler_fb35_mon_tuere_vo;
		sm_fehler_fb36_mon_tuere_hi := se_fehler_fb36_mon_tuere_hi;
		sm_fehler_fb37_mon_tuere_disk_vo := se_fehler_fb37_mon_tuere_disk_vo;
		sm_fehler_fb38_mon_tuere_disk_hi := se_fehler_fb38_mon_tuere_disk_hi;
		sm_fehler_fb39_mon_tuere_meld_vo := se_fehler_fb39_mon_tuere_meld_vo;
		sm_fehler_fb40_mon_tuere_meld_hi := se_fehler_fb40_mon_tuere_meld_hi;

		IF gst_datensatz.st_md.b_hublift_links_aktiv THEN
			sm_not_halt_hublift_links := NOT e_not_halt_hublift_links_ok;
		END_IF

		(*-----------------------Weiterschaltbedingungen----------------------------*)
		IF st_ctrl_in.b_quitt AND NOT fb_state_entry.E THEN
			st_ctrl_out.b_fehler := FALSE;
			fb_ton_quitt.IN := TRUE;
		END_IF

		IF fb_ton_quitt.Q THEN
			fb_ton_quitt.IN := FALSE;
			fb_state_entry.i16_next_step := INIT;
		END_IF
END_CASE

fb_state_entry(
	i16_next_step:= ,
	i16_pos:= 2,
	s_debugtext:= ,
	E=> ,
	X=> , 
	i16_step=> ,
	i16_last_step=> );

IF st_config.b_config_fertig THEN
	(* Fehlermeldungen und Betriebsmeldungen ab dem Startindex in die globalen Meldungsarrays schreiben *)
	garr_stoermeldungen[st_config.i16_meld_startindex + 0] := sm_steuerung_aus;
	garr_stoermeldungen[st_config.i16_meld_startindex + 1] := sm_not_halt_intern;
	garr_stoermeldungen[st_config.i16_meld_startindex + 2] := sm_not_halt_extern;
	garr_stoermeldungen[st_config.i16_meld_startindex + 3] := sm_tuere_vorne_offen;
	garr_stoermeldungen[st_config.i16_meld_startindex + 4] := sm_tuere_hinten_offen;
	garr_stoermeldungen[st_config.i16_meld_startindex + 5] := sm_tuere_vorne_diskrepanz;
	garr_stoermeldungen[st_config.i16_meld_startindex + 6] := sm_tuere_hinten_diskrepanz;
	garr_stoermeldungen[st_config.i16_meld_startindex + 7] := sm_bestueckachse_sto;
	garr_stoermeldungen[st_config.i16_meld_startindex + 8] := sm_bestueckachse_sls;
	garr_stoermeldungen[st_config.i16_meld_startindex + 9] := sm_z_achse_sto;
	garr_stoermeldungen[st_config.i16_meld_startindex + 10] := sm_z_achse_sls;
	garr_stoermeldungen[st_config.i16_meld_startindex + 11] := sm_y_achse_sto;
	garr_stoermeldungen[st_config.i16_meld_startindex + 12] := sm_y_achse_sls;
	garr_stoermeldungen[st_config.i16_meld_startindex + 13] := sm_not_halt_frontseite;
	garr_stoermeldungen[st_config.i16_meld_startindex + 14] := sm_not_halt_rueckseite;
	garr_stoermeldungen[st_config.i16_meld_startindex + 15] := sm_not_halt_bediengeraet;
	garr_stoermeldungen[st_config.i16_meld_startindex + 16] := sm_b_achse_sto;
	garr_stoermeldungen[st_config.i16_meld_startindex + 17] := sm_b_achse_sls;
	garr_stoermeldungen[st_config.i16_meld_startindex + 18] := sm_transport_achse_sto;
	garr_stoermeldungen[st_config.i16_meld_startindex + 19] := sm_transport_achse_sls;
	garr_stoermeldungen[st_config.i16_meld_startindex + 20] := sm_fehler_fb1_opmode;
	garr_stoermeldungen[st_config.i16_meld_startindex + 21] := sm_fehler_fb9_estop_nothalt_front;
	garr_stoermeldungen[st_config.i16_meld_startindex + 22] := sm_fehler_fb10_estop_nothalt_ext;
	garr_stoermeldungen[st_config.i16_meld_startindex + 23] := sm_fehler_fb15_edm_nothalt_ext	;
	garr_stoermeldungen[st_config.i16_meld_startindex + 24] := sm_fehler_fb16_edm_nothalt_schuetz;
	garr_stoermeldungen[st_config.i16_meld_startindex + 25] := sm_fehler_fb17_edm_ventilinsel;
	garr_stoermeldungen[st_config.i16_meld_startindex + 26] := sm_fehler_fb28_edm_foerderband;
	garr_stoermeldungen[st_config.i16_meld_startindex + 27] := sm_fehler_fb30_estop_rueck;
	garr_stoermeldungen[st_config.i16_meld_startindex + 28] := sm_fehler_fb31_estop_bedien;
	garr_stoermeldungen[st_config.i16_meld_startindex + 29] := sm_fehler_fb35_mon_tuere_vo;
	garr_stoermeldungen[st_config.i16_meld_startindex + 30] := sm_fehler_fb36_mon_tuere_hi;
	garr_stoermeldungen[st_config.i16_meld_startindex + 31] := sm_fehler_fb37_mon_tuere_disk_vo;
	garr_stoermeldungen[st_config.i16_meld_startindex + 32] := sm_fehler_fb38_mon_tuere_disk_hi;
	garr_stoermeldungen[st_config.i16_meld_startindex + 33] := sm_fehler_fb39_mon_tuere_meld_vo;
	garr_stoermeldungen[st_config.i16_meld_startindex + 34] := sm_fehler_fb40_mon_tuere_meld_hi;
	garr_stoermeldungen[st_config.i16_meld_startindex + 35] := sm_not_halt_hublift_links;
	garr_stoermeldungen[st_config.i16_meld_startindex + 36] := FALSE;
	garr_stoermeldungen[st_config.i16_meld_startindex + 37] := FALSE;
	garr_stoermeldungen[st_config.i16_meld_startindex + 38] := FALSE;
	garr_stoermeldungen[st_config.i16_meld_startindex + 39] := FALSE;

	garr_betriebsmeldungen[st_config.i16_meld_startindex + 0] := bm_taste_steuerung_ein_verhaengt;
	garr_betriebsmeldungen[st_config.i16_meld_startindex + 1] := bm_taste_steuerung_aus_verhaengt;
	garr_betriebsmeldungen[st_config.i16_meld_startindex + 2] := bm_taste_stoerung_quitt_verhaengt;
	garr_betriebsmeldungen[st_config.i16_meld_startindex + 3] := FALSE;
	garr_betriebsmeldungen[st_config.i16_meld_startindex + 4] := FALSE;
	garr_betriebsmeldungen[st_config.i16_meld_startindex + 5] := FALSE;
	garr_betriebsmeldungen[st_config.i16_meld_startindex + 6] := FALSE;
	garr_betriebsmeldungen[st_config.i16_meld_startindex + 7] := FALSE;
	garr_betriebsmeldungen[st_config.i16_meld_startindex + 8] := FALSE;
	garr_betriebsmeldungen[st_config.i16_meld_startindex + 9] := FALSE;
	garr_betriebsmeldungen[st_config.i16_meld_startindex + 10] := FALSE;
	garr_betriebsmeldungen[st_config.i16_meld_startindex + 11] := FALSE;
	garr_betriebsmeldungen[st_config.i16_meld_startindex + 12] := FALSE;
	garr_betriebsmeldungen[st_config.i16_meld_startindex + 13] := FALSE;
	garr_betriebsmeldungen[st_config.i16_meld_startindex + 14] := FALSE;
	garr_betriebsmeldungen[st_config.i16_meld_startindex + 15] := FALSE;
	garr_betriebsmeldungen[st_config.i16_meld_startindex + 16] := FALSE;
	garr_betriebsmeldungen[st_config.i16_meld_startindex + 17] := FALSE;
	garr_betriebsmeldungen[st_config.i16_meld_startindex + 18] := FALSE;
	garr_betriebsmeldungen[st_config.i16_meld_startindex + 19] := FALSE;
END_IF
END_PROGRAM

(* POU EPT Lib/Funktionen/F_Vergleich_LReal, ST *)
FUNCTION F_Vergleich_LReal : BOOL
VAR_INPUT
	lr_wert			: LREAL;
	lr_vergleichswert	: LREAL;
END_VAR
VAR
	lr_toleranz		: LREAL := 0.02;
END_VAR
IF ABS(lr_wert - lr_vergleichswert) < lr_toleranz THEN
	F_Vergleich_LReal := TRUE;
ELSE
	F_Vergleich_LReal := FALSE;
END_IF
END_FUNCTION

(* POU EPT Lib/Ethercat Diagnose/ST_EthercatDiag, ST *)
PROGRAM ST_EthercatDiag
VAR_INPUT
	st_config						: struct_config;
	st_ctrl_in						: struct_ctrl_in;
END_VAR
VAR_OUTPUT
	st_ctrl_out					: struct_ctrl_out;
END_VAR
VAR
	fb_ton_quitt					: TON;
	fb_ton_wz					: TON;
	fb_state_entry					: ST_StateEntry;
	fb_get_local_ams_netid		: ST_GetLocalAMSNetID;
	id							:  INT := 0;
	s_ec_slave_net_id			: ARRAY[0..8] OF  T_AmsNetId;
	arr_ec_slave_net_id			AT %I* : ARRAY[0..8] OF  T_AmsNetIdArr;

	sm_fehler_netid				: BOOL := FALSE;
END_VAR
fb_ton_quitt(IN:= , PT:= t#100ms, Q=> , ET=> );
fb_ton_wz(IN:= , PT:= t#10s , Q=> , ET=> );

fb_state_entry(
	i16_next_step:= ,
	i16_pos:= 1,
	s_debugtext:= ,
	E=> ,
	X=> ,
	i16_step=> ,
	i16_last_step=> );

CASE fb_state_entry.i16_step OF
(*=======================================================*)
	0:	(* Initialisierung *)
		st_ctrl_out.b_fehler := FALSE;
		st_ctrl_out.b_fertig := FALSE;
		st_ctrl_out.b_bereit := FALSE;
		fb_get_local_ams_netid.bExecute := FALSE;
		fb_get_local_ams_netid.bQuit := FALSE;
		sm_fehler_netid := FALSE;

		FOR id := 0  TO (SIZEOF (arr_ec_slave_net_id) / SIZEOF (arr_ec_slave_net_id[0]))-1 BY 1DO
			s_ec_slave_net_id[id] := '';
		END_FOR

		(*-----------------------Weiterschaltbedingungen----------------------------*)
		IF fb_get_local_ams_netid.bReady THEN
			fb_state_entry.i16_next_step := 10;
		END_IF

(*=======================================================*)
	10:	(* Die AMS-NetID des lokalen PC ermitteln *)
		IF fb_state_entry.E THEN
			fb_get_local_ams_netid.bExecute := TRUE;
		END_IF

		(*-----------------------Weiterschaltbedingungen----------------------------*)
		IF fb_get_local_ams_netid.bBusy THEN
			fb_get_local_ams_netid.bExecute := FALSE;
			fb_state_entry.i16_next_step := 20;
		END_IF

(*=======================================================*)
	20:

		(*-----------------------Weiterschaltbedingungen----------------------------*)
		IF NOT fb_get_local_ams_netid.bBusy  AND fb_get_local_ams_netid.bReady THEN
			IF NOT fb_get_local_ams_netid.bError THEN
				fb_state_entry.i16_next_step := 30;
			ELSE	(* Fehler *)
				sm_fehler_netid := TRUE;
				fb_state_entry.i16_next_step := FEHLER;
			END_IF
		END_IF

(*=======================================================*)
	30:	(* Umwandeln der Slave NetId von der Arrayform in die Stringform *)
		IF fb_state_entry.E THEN
			FOR id := 0  TO (SIZEOF (arr_ec_slave_net_id) / SIZEOF (arr_ec_slave_net_id[0]))-1 BY 1DO
				s_ec_slave_net_id[id] := F_CreateAmsNetId(nIds := arr_ec_slave_net_id[id]);
			END_FOR
		END_IF

		st_ctrl_out.b_fertig := TRUE;

(*=======================================================*)
	FEHLER: (* Fehler *)
		IF fb_state_entry.E THEN
			st_ctrl_out.b_fehler := TRUE;
			fb_ton_quitt.IN := FALSE;
			fb_get_local_ams_netid.bExecute := FALSE;
			fb_get_local_ams_netid.bQuit := FALSE;
		END_IF

		(*-----------------------Weiterschaltbedingungen----------------------------*)
		IF st_ctrl_in.b_quitt AND NOT fb_state_entry.E THEN
			st_ctrl_out.b_fehler := FALSE;
			fb_get_local_ams_netid .bQuit := TRUE;
			fb_ton_quitt.IN := TRUE;
		END_IF

		IF fb_ton_quitt.Q THEN
			fb_ton_quitt.IN := FALSE;
			fb_state_entry.i16_next_step := 0;
		END_IF
END_CASE

fb_state_entry(
	i16_next_step:= ,
	i16_pos:= 2,
	s_debugtext:= ,
	E=> ,
	X=> , 
	i16_step=> ,
	i16_last_step=> );

fb_get_local_ams_netid(
	bExecute:= , 
	bQuit:= , 
	bBusy=> , 
	bReady=> , 
	bError=> , 
	nErrId=> , 
	s_ams_netid=> );
END_PROGRAM

(* POU EPT Lib/Programmbausteine/Routing/ST_GetLocalAMSNetID, ST *)
FUNCTION_BLOCK ST_GetLocalAMSNetID
VAR_INPUT
	bExecute			: BOOL;
	bQuit				: BOOL;
END_VAR
VAR_OUTPUT
	bBusy				: BOOL;
	bReady				: BOOL;
	bError				: BOOL;
	nErrId				: UDINT;
	s_ams_netid			: T_AmsNetId;
END_VAR
VAR
	fb_ton_quitt					: TON;
	fb_state_entry					: ST_StateEntry;
	fb_r_trig_execute				: R_TRIG;
	fb_get_local_ams_netId		: FB_GetLocalAmsNetId;
	local_ams_netid				: T_AmsNetId := '0.0.0.0.0.0';
	ams_netid_arr				: T_AmsNetIdArr ;
END_VAR
fb_r_trig_execute(CLK:= bExecute, Q=> );
fb_ton_quitt(IN:= , PT:= t#100ms, Q=> , ET=> );

(* =======================================Toplevel========================================== *)
IF fb_state_entry.i16_next_step > INIT AND fb_state_entry.i16_next_step < FEHLER THEN
	 IF fb_get_local_ams_netId.bError THEN
		fb_state_entry.i16_next_step := FEHLER;
	END_IF
END_IF

fb_state_entry(
	i16_next_step:= ,
	i16_pos:= 1,
	s_debugtext:= ,
	E=> ,
	X=> ,
	i16_step=> ,
	i16_last_step=> );

CASE fb_state_entry.i16_step OF
(*=======================================================*)
	0:
		fb_state_entry.i16_next_step := INIT;

(*=======================================================*)
	10:(* INIT *)
		bBusy := FALSE;
		bReady := FALSE;
		bError := FALSE;
		nErrId := 0;
		s_ams_netid :=  '0.0.0.0.0.0';
		fb_get_local_ams_netId.bExecute := FALSE;
		fb_state_entry.i16_next_step := 20;

(*=======================================================*)
	20:	(* Warte auf Execute-Befehl *)
		IF fb_state_entry.E THEN
			bReady := TRUE;
		END_IF

		(*-----------------------Weiterschaltbedingungen----------------------------*)
		IF fb_r_trig_execute.Q THEN
			bReady := FALSE;
			bBusy := TRUE;
			fb_state_entry.i16_next_step := 30;
		END_IF

(*=======================================================*)
	30:	(* Starte mit Auslesen der NetID des lokalen PC *)
		IF fb_state_entry.E THEN
			fb_get_local_ams_netId.bExecute := TRUE;
		END_IF

		IF fb_get_local_ams_netId.bBusy THEN
			fb_get_local_ams_netId.bExecute := FALSE;
			fb_state_entry.i16_next_step := 40;
		END_IF

(*=======================================================*)
	40:	(* NetID wurde ausgelesen *)
		IF NOT fb_get_local_ams_netId.bBusy THEN
			IF NOT fb_get_local_ams_netId.bError THEN
				bBusy := FALSE;
				fb_state_entry.i16_next_step := 50;
			ELSE	(* Fehler *)
				fb_state_entry.i16_next_step := 1000;
			END_IF
		END_IF

(*=======================================================*)
	50:	(* Prüfe NetID  *)
		IF local_ams_netid <> '0.0.0.0.0.0' THEN
			s_ams_netid := local_ams_netid;
			fb_state_entry.i16_next_step := 999;
		ELSE	(* Fehler *)
			fb_state_entry.i16_next_step := 1000;
		END_IF

(*=======================================================*)
	999:	(* Kontrollschritt: NetID ist korrekt *)
		fb_state_entry.i16_next_step := 20;

(*=======================================================*)
	FEHLER: (* Fehler *)
		IF fb_state_entry.E THEN
			bBusy := FALSE;
			bReady := FALSE;
			bError := TRUE;
			fb_get_local_ams_netId.bExecute := FALSE;
			fb_ton_quitt.IN := FALSE;
		END_IF

		(*-----------------------Weiterschaltbedingungen----------------------------*)
		IF bQuit AND NOT fb_state_entry.E THEN
			bError := FALSE;
			fb_ton_quitt.IN := TRUE;
			(* Quittierflanke für FB *)
			fb_get_local_ams_netId.bExecute := TRUE;
		END_IF

		IF fb_ton_quitt.Q THEN
			fb_ton_quitt.IN := FALSE;
			fb_state_entry.i16_next_step := INIT;
		END_IF
END_CASE

fb_state_entry(
	i16_next_step:= , 
	i16_pos:= 2,
	s_debugtext:= ,
	E=> ,
	X=> ,
	i16_step=> ,
	i16_last_step=> );

fb_get_local_ams_netId(
	bExecute:= ,
	tTimeOut:= DEFAULT_ADS_TIMEOUT,
	bBusy=> ,
	bError=> , 
	nErrId=> nErrId,
	AddrString=> local_ams_netid,
	AddrBytes=> ams_netid_arr);
END_FUNCTION_BLOCK

(* POU EPT Lib/Programmbausteine/Routing/PC-Suche/ST_RoutingBackpanel, ST *)
PROGRAM ST_RoutingBackpanel
VAR_INPUT
	st_config						: struct_config;
	st_ctrl_in						: struct_ctrl_in;
END_VAR
VAR_OUTPUT
	st_ctrl_out					: struct_ctrl_out;
END_VAR
VAR
	fb_ton_wz					: TON;
	arr_read_routing_info			: ARRAY [0..31] OF ST_AmsRouteEntry;
	b_routing_station_gefunden		: BOOL;
	fb_add_route_entry			: FB_AddRouteEntry;
	fb_enum_route_entry			: FB_EnumRouteEntry;
	fb_ton_quitt					: TON;
	fb_state_entry					: ST_StateEntry;
	i16_eintrag					: INT := 0;
	b_ibn_start_routing			: BOOL := FALSE;
	fb_r_trig_ibn_start_routing		: R_TRIG;
	fb_ton_ibn_start_routing		: TON;
	s_backpanel_adresse			: STRING[255] := '';
	s_backpanel_netid			: STRING[255] := '';
	s_backpanel_name			: STRING[255] := '';
	s_temp_net_string				: STRING[255] := '';
	i16_temp_net_int				: INT := 0;
	s_temp_ip_string				: STRING[255] := '';
	i16_temp_ip_int				: INT := 0;
	s_temp_string_p11			: STRING[255] := '';
	s_temp_string_p12			: STRING[255] := '';
	s_temp_string_p13			: STRING[255] := '';
	fb_get_local_ams_netid		: ST_GetLocalAMSNetID;
	fb_get_adapters_info			: ST_GetAdaptersInfo;
	fb_get_host_name				: FB_GetHostName;
	fb_get_host_addr_by_name		: FB_GetHostAddrByName;
	st_pc_adapter_info			: ST_IpAdapterInfo;
	st_backpanel_adapter_info		: ST_IpAdapterInfo;
	sm_fehler_netid				: BOOL := FALSE;
	sm_fehler_adapter_info		: BOOL := FALSE;
	sm_fehler_host_name			: BOOL := FALSE;
	sm_fehler_host_addr			: BOOL := FALSE;
END_VAR
fb_ton_quitt(IN:= , PT:= t#100ms, Q=> , ET=> );
fb_ton_wz(IN:= , PT:= t#10s , Q=> , ET=> );

fb_r_trig_ibn_start_routing(CLK:= b_ibn_start_routing, Q=> );
fb_ton_ibn_start_routing(IN:= , PT:= t#1s, Q=> , ET=> );

IF fb_r_trig_ibn_start_routing.Q THEN
	fb_ton_ibn_start_routing.IN := TRUE;
ELSE
	IF fb_ton_ibn_start_routing.Q THEN
		b_ibn_start_routing := FALSE;
	 	fb_ton_ibn_start_routing.IN := FALSE;
	END_IF
END_IF

(* =======================================Toplevel========================================== *)
IF fb_state_entry.i16_next_step > INIT AND fb_state_entry.i16_next_step < FEHLER THEN
	 IF fb_get_adapters_info.bError OR fb_get_local_ams_netid.bError THEN
		fb_state_entry.i16_next_step := FEHLER;
	END_IF
END_IF

fb_state_entry(
	i16_next_step:= ,
	i16_pos:= 1,
	s_debugtext:= ,
	E=> ,
	X=> , 
	i16_step=> ,
	i16_last_step=> );

CASE fb_state_entry.i16_step OF
(*=======================================================*)
	0:
		fb_state_entry.i16_next_step := INIT;

